LIN {X 54.744,Y 107.989,Z 76.139,A 180.000,B 0.000,C 180.000} C_DIS
LIN {X 54.880,Y 108.068,Z 76.134,A 180.000,B 0.000,C 180.000} C_DIS
LIN {X 55.020,Y 108.140,Z 76.129,A 180.000,B 0.000,C 180.000} C_DIS
LIN {X 55.161,Y 108.210,Z 76.124,A 180.000,B 0.000,C 180.000} C_DIS
LIN {X 55.302,Y 108.281,Z 76.120,A 180.000,B 0.000,C 180.000} C_DIS
LIN {X 55.444,Y 108.349,Z 76.115,A 180.000,B 0.000,C 180.000} C_DIS
LIN {X 55.590,Y 108.409,Z 76.111,A 180.000,B 0.000,C 180.000} C_DIS
LIN {X 55.736,Y 108.467,Z 76.106,A 180.000,B 0.000,C 180.000} C_DIS
LIN {X 55.883,Y 108.525,Z 76.102,A 180.000,B 0.000,C 180.000} C_DIS
LIN {X 56.030,Y 108.581,Z 76.097,A 180.000,B 0.000,C 180.000} C_DIS
LIN {X 56.180,Y 108.630,Z 76.093,A 180.000,B 0.000,C 180.000} C_DIS
LIN {X 56.331,Y 108.674,Z 76.089,A 180.000,B 0.000,C 180.000} C_DIS
LIN {X 56.482,Y 108.719,Z 76.085,A 180.000,B 0.000,C 180.000} C_DIS
LIN {X 56.633,Y 108.763,Z 76.081,A 180.000,B 0.000,C 180.000} C_DIS
LIN {X 56.786,Y 108.800,Z 76.077,A 180.000,B 0.000,C 180.000} C_DIS
LIN {X 56.940,Y 108.831,Z 76.073,A 180.000,B 0.000,C 180.000} C_DIS
LIN {X 57.095,Y 108.863,Z 76.070,A 180.000,B 0.000,C 180.000} C_DIS
LIN {X 57.249,Y 108.894,Z 76.066,A 180.000,B 0.000,C 180.000} C_DIS
LIN {X 57.405,Y 108.919,Z 76.062,A 180.000,B 0.000,C 180.000} C_DIS
LIN {X 57.561,Y 108.937,Z 76.059,A 180.000,B 0.000,C 180.000} C_DIS
LIN {X 57.718,Y 108.954,Z 76.056,A 180.000,B 0.000,C 180.000} C_DIS
LIN {X 57.874,Y 108.972,Z 76.052,A 180.000,B 0.000,C 180.000} C_DIS
LIN {X 58.031,Y 108.985,Z 76.049,A 180.000,B 0.000,C 180.000} C_DIS
LIN {X 58.188,Y 108.990,Z 76.046,A 180.000,B 0.000,C 180.000} C_DIS
LIN {X 58.346,Y 108.994,Z 76.043,A 180.000,B 0.000,C 180.000} C_DIS
LIN {X 58.503,Y 108.997,Z 76.040,A 180.000,B 0.000,C 180.000} C_DIS
LIN {X 58.661,Y 108.998,Z 76.037,A 180.000,B 0.000,C 180.000} C_DIS
LIN {X 58.818,Y 108.991,Z 76.034,A 180.000,B 0.000,C 180.000} C_DIS
LIN {X 58.975,Y 108.980,Z 76.032,A 180.000,B 0.000,C 180.000} C_DIS
LIN {X 59.132,Y 108.970,Z 76.029,A 180.000,B 0.000,C 180.000} C_DIS
LIN {X 59.290,Y 108.958,Z 76.027,A 180.000,B 0.000,C 180.000} C_DIS
LIN {X 59.601,Y 108.914,Z 76.022,A 180.000,B 0.000,C 180.000} C_DIS
LIN {X 59.913,Y 108.865,Z 76.018,A 180.000,B 0.000,C 180.000} C_DIS
LIN {X 60.220,Y 108.796,Z 76.014,A 180.000,B 0.000,C 180.000} C_DIS
LIN {X 60.526,Y 108.720,Z 76.011,A 180.000,B 0.000,C 180.000} C_DIS
LIN {X 60.826,Y 108.626,Z 76.008,A 180.000,B 0.000,C 180.000} C_DIS
LIN {X 61.124,Y 108.523,Z 76.005,A 180.000,B 0.000,C 180.000} C_DIS
LIN {X 61.272,Y 108.469,Z 76.004,A 180.000,B 0.000,C 180.000} C_DIS
LIN {X 61.416,Y 108.406,Z 76.003,A 180.000,B 0.000,C 180.000} C_DIS
LIN {X 61.704,Y 108.278,Z 76.002,A 180.000,B 0.000,C 180.000} C_DIS
LIN {X 61.847,Y 108.212,Z 76.001,A 180.000,B 0.000,C 180.000} C_DIS
LIN {X 61.986,Y 108.138,Z 76.001,A 180.000,B 0.000,C 180.000} C_DIS
LIN {X 62.261,Y 107.984,Z 76.000,A 180.000,B 0.000,C 180.000} C_DIS
LIN {X 62.461,Y 107.866,Z 76.000,A 180.000,B 0.000,C 180.000} C_DIS
; Cutting Move Starts
LIN {X 62.562,Y 107.802,Z 76.000,A 180.000,B 0.000,C 180.000} C_DIS
LIN {X 62.825,Y 107.623,Z 76.000,A 180.000,B 0.000,C 180.000} C_DIS
LIN {X 62.930,Y 107.551,Z 76.000,A 180.000,B 0.000,C 180.000} C_DIS
LIN {X 63.071,Y 107.444,Z 76.000,A 180.000,B 0.000,C 180.000} C_DIS
LIN {X 63.109,Y 107.413,Z 76.000,A 180.000,B 0.000,C 180.000} C_DIS
LIN {X 63.290,Y 107.265,Z 76.000,A 180.000,B 0.000,C 180.000} C_DIS
LIN {X 63.467,Y 107.120,Z 76.000,A 180.000,B 0.000,C 180.000} C_DIS
LIN {X 63.504,Y 107.086,Z 76.000,A 180.000,B 0.000,C 180.000} C_DIS
LIN {X 63.645,Y 106.952,Z 76.000,A 180.000,B 0.000,C 180.000} C_DIS
LIN {X 63.873,Y 106.729,Z 76.000,A 180.000,B 0.000,C 180.000} C_DIS
LIN {X 64.003,Y 106.596,Z 76.000,A 180.000,B 0.000,C 180.000} C_DIS
LIN {X 64.043,Y 106.550,Z 76.000,A 180.000,B 0.000,C 180.000} C_DIS
LIN {X 64.196,Y 106.371,Z 76.000,A 180.000,B 0.000,C 180.000} C_DIS
LIN {X 64.349,Y 106.193,Z 76.000,A 180.000,B 0.000,C 180.000} C_DIS
LIN {X 64.360,Y 106.179,Z 76.000,A 180.000,B 0.000,C 180.000} C_DIS
LIN {X 64.487,Y 106.014,Z 76.000,A 180.000,B 0.000,C 180.000} C_DIS
LIN {X 64.718,Y 105.690,Z 76.000,A 180.000,B 0.000,C 180.000} C_DIS
LIN {X 64.742,Y 105.656,Z 76.000,A 180.000,B 0.000,C 180.000} C_DIS
LIN {X 64.856,Y 105.477,Z 76.000,A 180.000,B 0.000,C 180.000} C_DIS
LIN {X 65.075,Y 105.104,Z 76.000,A 180.000,B 0.000,C 180.000} C_DIS
LIN {X 65.163,Y 104.941,Z 76.000,A 180.000,B 0.000,C 180.000} C_DIS
LIN {X 65.248,Y 104.762,Z 76.000,A 180.000,B 0.000,C 180.000} C_DIS
LIN {X 65.333,Y 104.584,Z 76.000,A 180.000,B 0.000,C 180.000} C_DIS
LIN {X 65.415,Y 104.405,Z 76.000,A 180.000,B 0.000,C 180.000} C_DIS
LIN {X 65.433,Y 104.360,Z 76.000,A 180.000,B 0.000,C 180.000} C_DIS
LIN {X 65.483,Y 104.226,Z 76.000,A 180.000,B 0.000,C 180.000} C_DIS
LIN {X 65.549,Y 104.047,Z 76.000,A 180.000,B 0.000,C 180.000} C_DIS
LIN {X 65.612,Y 103.878,Z 76.000,A 180.000,B 0.000,C 180.000} C_DIS
LIN {X 65.615,Y 103.869,Z 76.000,A 180.000,B 0.000,C 180.000} C_DIS
LIN {X 65.672,Y 103.690,Z 76.000,A 180.000,B 0.000,C 180.000} C_DIS
LIN {X 65.720,Y 103.511,Z 76.000,A 180.000,B 0.000,C 180.000} C_DIS
LIN {X 65.791,Y 103.253,Z 76.000,A 180.000,B 0.000,C 180.000} C_DIS
LIN {X 65.815,Y 103.153,Z 76.000,A 180.000,B 0.000,C 180.000} C_DIS
LIN {X 65.850,Y 102.975,Z 76.000,A 180.000,B 0.000,C 180.000} C_DIS
LIN {X 65.914,Y 102.617,Z 76.000,A 180.000,B 0.000,C 180.000} C_DIS
LIN {X 65.941,Y 102.438,Z 76.000,A 180.000,B 0.000,C 180.000} C_DIS
LIN {X 65.957,Y 102.260,Z 76.000,A 180.000,B 0.000,C 180.000} C_DIS
LIN {X 65.973,Y 102.081,Z 76.000,A 180.000,B 0.000,C 180.000} C_DIS
LIN {X 65.989,Y 101.902,Z 76.000,A 180.000,B 0.000,C 180.000} C_DIS
LIN {X 65.995,Y 101.723,Z 76.000,A 180.000,B 0.000,C 180.000} C_DIS
LIN {X 65.995,Y 101.366,Z 76.000,A 180.000,B 0.000,C 180.000} C_DIS
LIN {X 65.993,Y 101.187,Z 76.000,A 180.000,B 0.000,C 180.000} C_DIS
LIN {X 65.981,Y 101.008,Z 76.000,A 180.000,B 0.000,C 180.000} C_DIS
LIN {X 65.949,Y 100.651,Z 76.000,A 180.000,B 0.000,C 180.000} C_DIS
LIN {X 65.929,Y 100.472,Z 76.000,A 180.000,B 0.000,C 180.000} C_DIS
LIN {X 65.898,Y 100.293,Z 76.000,A 180.000,B 0.000,C 180.000} C_DIS
LIN {X 65.866,Y 100.114,Z 76.000,A 180.000,B 0.000,C 180.000} C_DIS
LIN {X 65.834,Y 99.936,Z 76.000,A 180.000,B 0.000,C 180.000} C_DIS
LIN {X 65.793,Y 99.757,Z 76.000,A 180.000,B 0.000,C 180.000} C_DIS
LIN {X 65.791,Y 99.747,Z 76.000,A 180.000,B 0.000,C 180.000} C_DIS
LIN {X 65.696,Y 99.399,Z 76.000,A 180.000,B 0.000,C 180.000} C_DIS
LIN {X 65.645,Y 99.221,Z 76.000,A 180.000,B 0.000,C 180.000} C_DIS
LIN {X 65.612,Y 99.122,Z 76.000,A 180.000,B 0.000,C 180.000} C_DIS
LIN {X 65.582,Y 99.042,Z 76.000,A 180.000,B 0.000,C 180.000} C_DIS
LIN {X 65.516,Y 98.863,Z 76.000,A 180.000,B 0.000,C 180.000} C_DIS
LIN {X 65.450,Y 98.684,Z 76.000,A 180.000,B 0.000,C 180.000} C_DIS
LIN {X 65.433,Y 98.640,Z 76.000,A 180.000,B 0.000,C 180.000} C_DIS
LIN {X 65.375,Y 98.505,Z 76.000,A 180.000,B 0.000,C 180.000} C_DIS
LIN {X 65.290,Y 98.327,Z 76.000,A 180.000,B 0.000,C 180.000} C_DIS
LIN {X 65.206,Y 98.148,Z 76.000,A 180.000,B 0.000,C 180.000} C_DIS
LIN {X 65.117,Y 97.969,Z 76.000,A 180.000,B 0.000,C 180.000} C_DIS
LIN {X 65.075,Y 97.896,Z 76.000,A 180.000,B 0.000,C 180.000} C_DIS
LIN {X 64.897,Y 97.592,Z 76.000,A 180.000,B 0.000,C 180.000} C_DIS
LIN {X 64.801,Y 97.433,Z 76.000,A 180.000,B 0.000,C 180.000} C_DIS
LIN {X 64.718,Y 97.310,Z 76.000,A 180.000,B 0.000,C 180.000} C_DIS
LIN {X 64.539,Y 97.060,Z 76.000,A 180.000,B 0.000,C 180.000} C_DIS
LIN {X 64.421,Y 96.897,Z 76.000,A 180.000,B 0.000,C 180.000} C_DIS
LIN {X 64.360,Y 96.821,Z 76.000,A 180.000,B 0.000,C 180.000} C_DIS
LIN {X 64.272,Y 96.718,Z 76.000,A 180.000,B 0.000,C 180.000} C_DIS
LIN {X 64.119,Y 96.539,Z 76.000,A 180.000,B 0.000,C 180.000} C_DIS
LIN {X 64.003,Y 96.404,Z 76.000,A 180.000,B 0.000,C 180.000} C_DIS
LIN {X 63.962,Y 96.360,Z 76.000,A 180.000,B 0.000,C 180.000} C_DIS
LIN {X 63.824,Y 96.223,Z 76.000,A 180.000,B 0.000,C 180.000} C_DIS
LIN {X 63.599,Y 96.003,Z 76.000,A 180.000,B 0.000,C 180.000} C_DIS
LIN {X 63.467,Y 95.880,Z 76.000,A 180.000,B 0.000,C 180.000} C_DIS
LIN {X 63.399,Y 95.824,Z 76.000,A 180.000,B 0.000,C 180.000} C_DIS
LIN {X 63.109,Y 95.587,Z 76.000,A 180.000,B 0.000,C 180.000} C_DIS
LIN {X 62.954,Y 95.466,Z 76.000,A 180.000,B 0.000,C 180.000} C_DIS
LIN {X 62.930,Y 95.449,Z 76.000,A 180.000,B 0.000,C 180.000} C_DIS
LIN {X 62.751,Y 95.327,Z 76.000,A 180.000,B 0.000,C 180.000} C_DIS
LIN {X 62.573,Y 95.206,Z 76.000,A 180.000,B 0.000,C 180.000} C_DIS
LIN {X 62.425,Y 95.109,Z 76.000,A 180.000,B 0.000,C 180.000} C_DIS
LIN {X 62.394,Y 95.091,Z 76.000,A 180.000,B 0.000,C 180.000} C_DIS
LIN {X 62.215,Y 94.990,Z 76.000,A 180.000,B 0.000,C 180.000} C_DIS
LIN {X 62.036,Y 94.890,Z 76.000,A 180.000,B 0.000,C 180.000} C_DIS
LIN {X 61.858,Y 94.794,Z 76.000,A 180.000,B 0.000,C 180.000} C_DIS
LIN {X 61.769,Y 94.751,Z 76.000,A 180.000,B 0.000,C 180.000} C_DIS
LIN {X 61.679,Y 94.711,Z 76.000,A 180.000,B 0.000,C 180.000} C_DIS
LIN {X 61.369,Y 94.573,Z 76.000,A 180.000,B 0.000,C 180.000} C_DIS
LIN {X 61.321,Y 94.552,Z 76.000,A 180.000,B 0.000,C 180.000} C_DIS
LIN {X 61.143,Y 94.483,Z 76.000,A 180.000,B 0.000,C 180.000} C_DIS
LIN {X 60.785,Y 94.360,Z 76.000,A 180.000,B 0.000,C 180.000} C_DIS
LIN {X 60.606,Y 94.302,Z 76.000,A 180.000,B 0.000,C 180.000} C_DIS
LIN {X 60.427,Y 94.256,Z 76.000,A 180.000,B 0.000,C 180.000} C_DIS
LIN {X 60.249,Y 94.212,Z 76.000,A 180.000,B 0.000,C 180.000} C_DIS
LIN {X 60.070,Y 94.167,Z 76.000,A 180.000,B 0.000,C 180.000} C_DIS
LIN {X 59.891,Y 94.131,Z 76.000,A 180.000,B 0.000,C 180.000} C_DIS
LIN {X 59.712,Y 94.103,Z 76.000,A 180.000,B 0.000,C 180.000} C_DIS
LIN {X 59.534,Y 94.075,Z 76.000,A 180.000,B 0.000,C 180.000} C_DIS
LIN {X 59.355,Y 94.049,Z 76.000,A 180.000,B 0.000,C 180.000} C_DIS
LIN {X 59.220,Y 94.036,Z 76.000,A 180.000,B 0.000,C 180.000} C_DIS
LIN {X 58.819,Y 94.010,Z 76.000,A 180.000,B 0.000,C 180.000} C_DIS
LIN {X 58.640,Y 94.001,Z 76.000,A 180.000,B 0.000,C 180.000} C_DIS
LIN {X 58.461,Y 94.004,Z 76.000,A 180.000,B 0.000,C 180.000} C_DIS
LIN {X 58.282,Y 94.008,Z 76.000,A 180.000,B 0.000,C 180.000} C_DIS
LIN {X 58.103,Y 94.012,Z 76.000,A 180.000,B 0.000,C 180.000} C_DIS
LIN {X 57.925,Y 94.023,Z 76.000,A 180.000,B 0.000,C 180.000} C_DIS
LIN {X 57.803,Y 94.036,Z 76.000,A 180.000,B 0.000,C 180.000} C_DIS
LIN {X 57.567,Y 94.062,Z 76.000,A 180.000,B 0.000,C 180.000} C_DIS
LIN {X 57.388,Y 94.083,Z 76.000,A 180.000,B 0.000,C 180.000} C_DIS
LIN {X 57.210,Y 94.114,Z 76.000,A 180.000,B 0.000,C 180.000} C_DIS
LIN {X 56.852,Y 94.186,Z 76.000,A 180.000,B 0.000,C 180.000} C_DIS
LIN {X 56.717,Y 94.215,Z 76.000,A 180.000,B 0.000,C 180.000} C_DIS
LIN {X 56.673,Y 94.226,Z 76.000,A 180.000,B 0.000,C 180.000} C_DIS
LIN {X 56.495,Y 94.277,Z 76.000,A 180.000,B 0.000,C 180.000} C_DIS
LIN {X 56.316,Y 94.330,Z 76.000,A 180.000,B 0.000,C 180.000} C_DIS
LIN {X 56.137,Y 94.383,Z 76.000,A 180.000,B 0.000,C 180.000} C_DIS
LIN {X 56.103,Y 94.394,Z 76.000,A 180.000,B 0.000,C 180.000} C_DIS
LIN {X 55.958,Y 94.445,Z 76.000,A 180.000,B 0.000,C 180.000} C_DIS
LIN {X 55.601,Y 94.587,Z 76.000,A 180.000,B 0.000,C 180.000} C_DIS
LIN {X 55.422,Y 94.661,Z 76.000,A 180.000,B 0.000,C 180.000} C_DIS
LIN {X 55.243,Y 94.749,Z 76.000,A 180.000,B 0.000,C 180.000} C_DIS
LIN {X 55.064,Y 94.838,Z 76.000,A 180.000,B 0.000,C 180.000} C_DIS
LIN {X 54.886,Y 94.929,Z 76.000,A 180.000,B 0.000,C 180.000} C_DIS
LIN {X 54.883,Y 94.930,Z 76.000,A 180.000,B 0.000,C 180.000} C_DIS
LIN {X 54.707,Y 95.033,Z 76.000,A 180.000,B 0.000,C 180.000} C_DIS
LIN {X 54.528,Y 95.144,Z 76.000,A 180.000,B 0.000,C 180.000} C_DIS
LIN {X 54.349,Y 95.254,Z 76.000,A 180.000,B 0.000,C 180.000} C_DIS
LIN {X 54.298,Y 95.288,Z 76.000,A 180.000,B 0.000,C 180.000} C_DIS
LIN {X 54.171,Y 95.379,Z 76.000,A 180.000,B 0.000,C 180.000} C_DIS
LIN {X 53.992,Y 95.512,Z 76.000,A 180.000,B 0.000,C 180.000} C_DIS
LIN {X 53.814,Y 95.645,Z 76.000,A 180.000,B 0.000,C 180.000} C_DIS
LIN {X 53.813,Y 95.646,Z 76.000,A 180.000,B 0.000,C 180.000} C_DIS
LIN {X 53.634,Y 95.796,Z 76.000,A 180.000,B 0.000,C 180.000} C_DIS
LIN {X 53.404,Y 96.003,Z 76.000,A 180.000,B 0.000,C 180.000} C_DIS
LIN {X 53.277,Y 96.118,Z 76.000,A 180.000,B 0.000,C 180.000} C_DIS
LIN {X 53.213,Y 96.181,Z 76.000,A 180.000,B 0.000,C 180.000} C_DIS
LIN {X 53.098,Y 96.303,Z 76.000,A 180.000,B 0.000,C 180.000} C_DIS
LIN {X 52.877,Y 96.539,Z 76.000,A 180.000,B 0.000,C 180.000} C_DIS
LIN {X 52.740,Y 96.698,Z 76.000,A 180.000,B 0.000,C 180.000} C_DIS
LIN {X 52.725,Y 96.718,Z 76.000,A 180.000,B 0.000,C 180.000} C_DIS
LIN {X 52.562,Y 96.927,Z 76.000,A 180.000,B 0.000,C 180.000} C_DIS
LIN {X 52.446,Y 97.075,Z 76.000,A 180.000,B 0.000,C 180.000} C_DIS
LIN {X 52.383,Y 97.161,Z 76.000,A 180.000,B 0.000,C 180.000} C_DIS
LIN {X 52.320,Y 97.254,Z 76.000,A 180.000,B 0.000,C 180.000} C_DIS
LIN {X 52.088,Y 97.612,Z 76.000,A 180.000,B 0.000,C 180.000} C_DIS
LIN {X 52.025,Y 97.715,Z 76.000,A 180.000,B 0.000,C 180.000} C_DIS
LIN {X 51.983,Y 97.790,Z 76.000,A 180.000,B 0.000,C 180.000} C_DIS
LIN {X 51.889,Y 97.969,Z 76.000,A 180.000,B 0.000,C 180.000} C_DIS
LIN {X 51.794,Y 98.148,Z 76.000,A 180.000,B 0.000,C 180.000} C_DIS
LIN {X 51.705,Y 98.327,Z 76.000,A 180.000,B 0.000,C 180.000} C_DIS
LIN {X 51.668,Y 98.412,Z 76.000,A 180.000,B 0.000,C 180.000} C_DIS
LIN {X 51.553,Y 98.684,Z 76.000,A 180.000,B 0.000,C 180.000} C_DIS
LIN {X 51.489,Y 98.838,Z 76.000,A 180.000,B 0.000,C 180.000} C_DIS
LIN {X 51.479,Y 98.863,Z 76.000,A 180.000,B 0.000,C 180.000} C_DIS
LIN {X 51.417,Y 99.042,Z 76.000,A 180.000,B 0.000,C 180.000} C_DIS
LIN {X 51.303,Y 99.399,Z 76.000,A 180.000,B 0.000,C 180.000} C_DIS
LIN {X 51.251,Y 99.578,Z 76.000,A 180.000,B 0.000,C 180.000} C_DIS
LIN {X 51.210,Y 99.757,Z 76.000,A 180.000,B 0.000,C 180.000} C_DIS
LIN {X 51.170,Y 99.936,Z 76.000,A 180.000,B 0.000,C 180.000} C_DIS
LIN {X 51.131,Y 100.106,Z 76.000,A 180.000,B 0.000,C 180.000} C_DIS
LIN {X 51.130,Y 100.114,Z 76.000,A 180.000,B 0.000,C 180.000} C_DIS
LIN {X 51.100,Y 100.293,Z 76.000,A 180.000,B 0.000,C 180.000} C_DIS
LIN {X 51.052,Y 100.651,Z 76.000,A 180.000,B 0.000,C 180.000} C_DIS
LIN {X 51.030,Y 100.829,Z 76.000,A 180.000,B 0.000,C 180.000} C_DIS
LIN {X 51.019,Y 101.008,Z 76.000,A 180.000,B 0.000,C 180.000} C_DIS
LIN {X 51.003,Y 101.366,Z 76.000,A 180.000,B 0.000,C 180.000} C_DIS
LIN {X 51.000,Y 101.545,Z 76.000,A 180.000,B 0.000,C 180.000} C_DIS
LIN {X 51.007,Y 101.723,Z 76.000,A 180.000,B 0.000,C 180.000} C_DIS
LIN {X 51.015,Y 101.902,Z 76.000,A 180.000,B 0.000,C 180.000} C_DIS
LIN {X 51.023,Y 102.081,Z 76.000,A 180.000,B 0.000,C 180.000} C_DIS
LIN {X 51.040,Y 102.260,Z 76.000,A 180.000,B 0.000,C 180.000} C_DIS
LIN {X 51.064,Y 102.438,Z 76.000,A 180.000,B 0.000,C 180.000} C_DIS
LIN {X 51.088,Y 102.617,Z 76.000,A 180.000,B 0.000,C 180.000} C_DIS
LIN {X 51.113,Y 102.796,Z 76.000,A 180.000,B 0.000,C 180.000} C_DIS
LIN {X 51.131,Y 102.894,Z 76.000,A 180.000,B 0.000,C 180.000} C_DIS
LIN {X 51.149,Y 102.975,Z 76.000,A 180.000,B 0.000,C 180.000} C_DIS
LIN {X 51.230,Y 103.332,Z 76.000,A 180.000,B 0.000,C 180.000} C_DIS
LIN {X 51.275,Y 103.511,Z 76.000,A 180.000,B 0.000,C 180.000} C_DIS
LIN {X 51.310,Y 103.624,Z 76.000,A 180.000,B 0.000,C 180.000} C_DIS
LIN {X 51.388,Y 103.869,Z 76.000,A 180.000,B 0.000,C 180.000} C_DIS
LIN {X 51.446,Y 104.047,Z 76.000,A 180.000,B 0.000,C 180.000} C_DIS
LIN {X 51.489,Y 104.162,Z 76.000,A 180.000,B 0.000,C 180.000} C_DIS
LIN {X 51.515,Y 104.226,Z 76.000,A 180.000,B 0.000,C 180.000} C_DIS
LIN {X 51.668,Y 104.588,Z 76.000,A 180.000,B 0.000,C 180.000} C_DIS
LIN {X 51.747,Y 104.762,Z 76.000,A 180.000,B 0.000,C 180.000} C_DIS
LIN {X 51.841,Y 104.941,Z 76.000,A 180.000,B 0.000,C 180.000} C_DIS
LIN {X 51.936,Y 105.120,Z 76.000,A 180.000,B 0.000,C 180.000} C_DIS
LIN {X 52.025,Y 105.285,Z 76.000,A 180.000,B 0.000,C 180.000} C_DIS
LIN {X 52.033,Y 105.299,Z 76.000,A 180.000,B 0.000,C 180.000} C_DIS
LIN {X 52.146,Y 105.477,Z 76.000,A 180.000,B 0.000,C 180.000} C_DIS
LIN {X 52.262,Y 105.656,Z 76.000,A 180.000,B 0.000,C 180.000} C_DIS
LIN {X 52.380,Y 105.835,Z 76.000,A 180.000,B 0.000,C 180.000} C_DIS
LIN {X 52.383,Y 105.839,Z 76.000,A 180.000,B 0.000,C 180.000} C_DIS
LIN {X 52.515,Y 106.014,Z 76.000,A 180.000,B 0.000,C 180.000} C_DIS
LIN {X 52.655,Y 106.193,Z 76.000,A 180.000,B 0.000,C 180.000} C_DIS
LIN {X 52.740,Y 106.302,Z 76.000,A 180.000,B 0.000,C 180.000} C_DIS
LIN {X 52.797,Y 106.371,Z 76.000,A 180.000,B 0.000,C 180.000} C_DIS
LIN {X 52.919,Y 106.506,Z 76.000,A 180.000,B 0.000,C 180.000} C_DIS
LIN {X 53.128,Y 106.729,Z 76.000,A 180.000,B 0.000,C 180.000} C_DIS
LIN {X 53.277,Y 106.882,Z 76.000,A 180.000,B 0.000,C 180.000} C_DIS
LIN {X 53.304,Y 106.908,Z 76.000,A 180.000,B 0.000,C 180.000} C_DIS
LIN {X 53.455,Y 107.044,Z 76.000,A 180.000,B 0.000,C 180.000} C_DIS
LIN {X 53.634,Y 107.204,Z 76.000,A 180.000,B 0.000,C 180.000} C_DIS
LIN {X 53.704,Y 107.265,Z 76.000,A 180.000,B 0.000,C 180.000} C_DIS
LIN {X 53.813,Y 107.354,Z 76.000,A 180.000,B 0.000,C 180.000} C_DIS
LIN {X 53.933,Y 107.444,Z 76.000,A 180.000,B 0.000,C 180.000} C_DIS
LIN {X 54.172,Y 107.623,Z 76.000,A 180.000,B 0.000,C 180.000} C_DIS
LIN {X 54.349,Y 107.746,Z 76.000,A 180.000,B 0.000,C 180.000} C_DIS
LIN {X 54.439,Y 107.802,Z 76.000,A 180.000,B 0.000,C 180.000} C_DIS
LIN {X 54.729,Y 107.980,Z 76.000,A 180.000,B 0.000,C 180.000} C_DIS
LIN {X 54.886,Y 108.071,Z 76.000,A 180.000,B 0.000,C 180.000} C_DIS
LIN {X 55.059,Y 108.159,Z 76.000,A 180.000,B 0.000,C 180.000} C_DIS
LIN {X 55.243,Y 108.251,Z 76.000,A 180.000,B 0.000,C 180.000} C_DIS
LIN {X 55.419,Y 108.338,Z 76.000,A 180.000,B 0.000,C 180.000} C_DIS
LIN {X 55.422,Y 108.339,Z 76.000,A 180.000,B 0.000,C 180.000} C_DIS
LIN {X 55.601,Y 108.413,Z 76.000,A 180.000,B 0.000,C 180.000} C_DIS
LIN {X 55.862,Y 108.517,Z 76.000,A 180.000,B 0.000,C 180.000} C_DIS
LIN {X 55.958,Y 108.555,Z 76.000,A 180.000,B 0.000,C 180.000} C_DIS
LIN {X 56.137,Y 108.617,Z 76.000,A 180.000,B 0.000,C 180.000} C_DIS
LIN {X 56.316,Y 108.670,Z 76.000,A 180.000,B 0.000,C 180.000} C_DIS
LIN {X 56.495,Y 108.723,Z 76.000,A 180.000,B 0.000,C 180.000} C_DIS
LIN {X 56.673,Y 108.774,Z 76.000,A 180.000,B 0.000,C 180.000} C_DIS
LIN {X 56.852,Y 108.814,Z 76.000,A 180.000,B 0.000,C 180.000} C_DIS
LIN {X 57.210,Y 108.886,Z 76.000,A 180.000,B 0.000,C 180.000} C_DIS
LIN {X 57.388,Y 108.917,Z 76.000,A 180.000,B 0.000,C 180.000} C_DIS
LIN {X 57.567,Y 108.938,Z 76.000,A 180.000,B 0.000,C 180.000} C_DIS
LIN {X 57.746,Y 108.957,Z 76.000,A 180.000,B 0.000,C 180.000} C_DIS
LIN {X 57.925,Y 108.977,Z 76.000,A 180.000,B 0.000,C 180.000} C_DIS
LIN {X 58.103,Y 108.988,Z 76.000,A 180.000,B 0.000,C 180.000} C_DIS
LIN {X 58.282,Y 108.992,Z 76.000,A 180.000,B 0.000,C 180.000} C_DIS
LIN {X 58.461,Y 108.996,Z 76.000,A 180.000,B 0.000,C 180.000} C_DIS
LIN {X 58.640,Y 108.999,Z 76.000,A 180.000,B 0.000,C 180.000} C_DIS
LIN {X 58.819,Y 108.990,Z 76.000,A 180.000,B 0.000,C 180.000} C_DIS
LIN {X 59.176,Y 108.967,Z 76.000,A 180.000,B 0.000,C 180.000} C_DIS
LIN {X 59.355,Y 108.951,Z 76.000,A 180.000,B 0.000,C 180.000} C_DIS
LIN {X 59.534,Y 108.925,Z 76.000,A 180.000,B 0.000,C 180.000} C_DIS
LIN {X 59.856,Y 108.874,Z 76.000,A 180.000,B 0.000,C 180.000} C_DIS
LIN {X 59.891,Y 108.869,Z 76.000,A 180.000,B 0.000,C 180.000} C_DIS
LIN {X 60.070,Y 108.833,Z 76.000,A 180.000,B 0.000,C 180.000} C_DIS
LIN {X 60.249,Y 108.788,Z 76.000,A 180.000,B 0.000,C 180.000} C_DIS
LIN {X 60.427,Y 108.744,Z 76.000,A 180.000,B 0.000,C 180.000} C_DIS
LIN {X 60.606,Y 108.698,Z 76.000,A 180.000,B 0.000,C 180.000} C_DIS
LIN {X 60.616,Y 108.695,Z 76.000,A 180.000,B 0.000,C 180.000} C_DIS
LIN {X 60.785,Y 108.640,Z 76.000,A 180.000,B 0.000,C 180.000} C_DIS
LIN {X 61.144,Y 108.517,Z 76.000,A 180.000,B 0.000,C 180.000} C_DIS
LIN {X 61.321,Y 108.448,Z 76.000,A 180.000,B 0.000,C 180.000} C_DIS
LIN {X 61.500,Y 108.369,Z 76.000,A 180.000,B 0.000,C 180.000} C_DIS
LIN {X 61.679,Y 108.289,Z 76.000,A 180.000,B 0.000,C 180.000} C_DIS
LIN {X 61.858,Y 108.206,Z 76.000,A 180.000,B 0.000,C 180.000} C_DIS
LIN {X 61.948,Y 108.159,Z 76.000,A 180.000,B 0.000,C 180.000} C_DIS
LIN {X 62.036,Y 108.110,Z 76.000,A 180.000,B 0.000,C 180.000} C_DIS
LIN {X 62.268,Y 107.980,Z 76.000,A 180.000,B 0.000,C 180.000} C_DIS
LIN {X 62.394,Y 107.909,Z 76.000,A 180.000,B 0.000,C 180.000} C_DIS
LIN {X 62.461,Y 107.866,Z 76.000,A 180.000,B 0.000,C 180.000} C_DIS
; Link Move Starts
LIN {X 62.724,Y 107.692,Z 76.000,A 180.000,B 0.000,C 180.000} C_DIS
LIN {X 62.983,Y 107.513,Z 75.999,A 180.000,B 0.000,C 180.000} C_DIS
LIN {X 63.228,Y 107.315,Z 75.998,A 180.000,B 0.000,C 180.000} C_DIS
LIN {X 63.472,Y 107.115,Z 75.996,A 180.000,B 0.000,C 180.000} C_DIS
LIN {X 63.700,Y 106.898,Z 75.994,A 180.000,B 0.000,C 180.000} C_DIS
LIN {X 63.925,Y 106.678,Z 75.991,A 180.000,B 0.000,C 180.000} C_DIS
LIN {X 64.135,Y 106.443,Z 75.988,A 180.000,B 0.000,C 180.000} C_DIS
LIN {X 64.340,Y 106.204,Z 75.985,A 180.000,B 0.000,C 180.000} C_DIS
LIN {X 64.438,Y 106.081,Z 75.983,A 180.000,B 0.000,C 180.000} C_DIS
LIN {X 64.530,Y 105.953,Z 75.981,A 180.000,B 0.000,C 180.000} C_DIS
LIN {X 64.713,Y 105.697,Z 75.977,A 180.000,B 0.000,C 180.000} C_DIS
LIN {X 64.802,Y 105.566,Z 75.974,A 180.000,B 0.000,C 180.000} C_DIS
LIN {X 64.883,Y 105.431,Z 75.972,A 180.000,B 0.000,C 180.000} C_DIS
LIN {X 64.963,Y 105.296,Z 75.969,A 180.000,B 0.000,C 180.000} C_DIS
LIN {X 65.043,Y 105.160,Z 75.967,A 180.000,B 0.000,C 180.000} C_DIS
LIN {X 65.121,Y 105.023,Z 75.964,A 180.000,B 0.000,C 180.000} C_DIS
LIN {X 65.191,Y 104.882,Z 75.961,A 180.000,B 0.000,C 180.000} C_DIS
LIN {X 65.259,Y 104.740,Z 75.959,A 180.000,B 0.000,C 180.000} C_DIS
LIN {X 65.326,Y 104.598,Z 75.956,A 180.000,B 0.000,C 180.000} C_DIS
LIN {X 65.393,Y 104.455,Z 75.952,A 180.000,B 0.000,C 180.000} C_DIS
LIN {X 65.452,Y 104.309,Z 75.949,A 180.000,B 0.000,C 180.000} C_DIS
LIN {X 65.507,Y 104.161,Z 75.946,A 180.000,B 0.000,C 180.000} C_DIS
LIN {X 65.562,Y 104.014,Z 75.943,A 180.000,B 0.000,C 180.000} C_DIS
LIN {X 65.616,Y 103.866,Z 75.939,A 180.000,B 0.000,C 180.000} C_DIS
LIN {X 65.664,Y 103.716,Z 75.936,A 180.000,B 0.000,C 180.000} C_DIS
LIN {X 65.706,Y 103.564,Z 75.932,A 180.000,B 0.000,C 180.000} C_DIS
LIN {X 65.747,Y 103.412,Z 75.928,A 180.000,B 0.000,C 180.000} C_DIS
LIN {X 65.789,Y 103.260,Z 75.925,A 180.000,B 0.000,C 180.000} C_DIS
LIN {X 65.826,Y 103.107,Z 75.921,A 180.000,B 0.000,C 180.000} C_DIS
LIN {X 65.854,Y 102.952,Z 75.917,A 180.000,B 0.000,C 180.000} C_DIS
LIN {X 65.882,Y 102.797,Z 75.913,A 180.000,B 0.000,C 180.000} C_DIS
LIN {X 65.910,Y 102.642,Z 75.909,A 180.000,B 0.000,C 180.000} C_DIS
LIN {X 65.935,Y 102.487,Z 75.905,A 180.000,B 0.000,C 180.000} C_DIS
LIN {X 65.951,Y 102.330,Z 75.900,A 180.000,B 0.000,C 180.000} C_DIS
LIN {X 65.965,Y 102.173,Z 75.896,A 180.000,B 0.000,C 180.000} C_DIS
LIN {X 65.979,Y 102.016,Z 75.892,A 180.000,B 0.000,C 180.000} C_DIS
LIN {X 65.991,Y 101.859,Z 75.887,A 180.000,B 0.000,C 180.000} C_DIS
LIN {X 65.995,Y 101.702,Z 75.883,A 180.000,B 0.000,C 180.000} C_DIS
LIN {X 65.995,Y 101.544,Z 75.878,A 180.000,B 0.000,C 180.000} C_DIS
LIN {X 65.995,Y 101.387,Z 75.873,A 180.000,B 0.000,C 180.000} C_DIS
LIN {X 65.995,Y 101.229,Z 75.869,A 180.000,B 0.000,C 180.000} C_DIS
LIN {X 65.987,Y 101.072,Z 75.864,A 180.000,B 0.000,C 180.000} C_DIS
LIN {X 65.973,Y 100.915,Z 75.859,A 180.000,B 0.000,C 180.000} C_DIS
LIN {X 65.959,Y 100.758,Z 75.854,A 180.000,B 0.000,C 180.000} C_DIS
LIN {X 65.952,Y 100.680,Z 75.851,A 180.000,B 0.000,C 180.000} C_DIS
LIN {X 65.945,Y 100.601,Z 75.849,A 180.000,B 0.000,C 180.000} C_DIS
LIN {X 65.936,Y 100.523,Z 75.846,A 180.000,B 0.000,C 180.000} C_DIS
LIN {X 65.925,Y 100.445,Z 75.844,A 180.000,B 0.000,C 180.000} C_DIS
LIN {X 65.911,Y 100.367,Z 75.841,A 180.000,B 0.000,C 180.000} C_DIS
LIN {X 65.898,Y 100.290,Z 75.839,A 180.000,B 0.000,C 180.000} C_DIS
LIN {X 65.884,Y 100.212,Z 75.836,A 180.000,B 0.000,C 180.000} C_DIS
LIN {X 65.856,Y 100.057,Z 75.831,A 180.000,B 0.000,C 180.000} C_DIS
LIN {X 65.842,Y 99.980,Z 75.828,A 180.000,B 0.000,C 180.000} C_DIS
LIN {X 65.828,Y 99.902,Z 75.825,A 180.000,B 0.000,C 180.000} C_DIS
LIN {X 65.811,Y 99.825,Z 75.823,A 180.000,B 0.000,C 180.000} C_DIS
LIN {X 65.791,Y 99.749,Z 75.820,A 180.000,B 0.000,C 180.000} C_DIS
LIN {X 65.750,Y 99.597,Z 75.815,A 180.000,B 0.000,C 180.000} C_DIS
LIN {X 65.709,Y 99.445,Z 75.809,A 180.000,B 0.000,C 180.000} C_DIS
LIN {X 65.688,Y 99.369,Z 75.807,A 180.000,B 0.000,C 180.000} C_DIS
LIN {X 65.667,Y 99.293,Z 75.804,A 180.000,B 0.000,C 180.000} C_DIS
LIN {X 65.644,Y 99.218,Z 75.801,A 180.000,B 0.000,C 180.000} C_DIS
LIN {X 65.619,Y 99.143,Z 75.798,A 180.000,B 0.000,C 180.000} C_DIS
LIN {X 65.592,Y 99.069,Z 75.796,A 180.000,B 0.000,C 180.000} C_DIS
LIN {X 65.538,Y 98.921,Z 75.790,A 180.000,B 0.000,C 180.000} C_DIS
LIN {X 65.456,Y 98.700,Z 75.782,A 180.000,B 0.000,C 180.000} C_DIS
LIN {X 65.427,Y 98.626,Z 75.779,A 180.000,B 0.000,C 180.000} C_DIS
LIN {X 65.397,Y 98.554,Z 75.776,A 180.000,B 0.000,C 180.000} C_DIS
LIN {X 65.364,Y 98.482,Z 75.774,A 180.000,B 0.000,C 180.000} C_DIS
LIN {X 65.297,Y 98.340,Z 75.768,A 180.000,B 0.000,C 180.000} C_DIS
LIN {X 65.195,Y 98.126,Z 75.760,A 180.000,B 0.000,C 180.000} C_DIS
LIN {X 65.161,Y 98.055,Z 75.757,A 180.000,B 0.000,C 180.000} C_DIS
LIN {X 65.125,Y 97.985,Z 75.754,A 180.000,B 0.000,C 180.000} C_DIS
LIN {X 65.087,Y 97.916,Z 75.752,A 180.000,B 0.000,C 180.000} C_DIS
LIN {X 65.048,Y 97.848,Z 75.749,A 180.000,B 0.000,C 180.000} C_DIS
LIN {X 64.968,Y 97.713,Z 75.743,A 180.000,B 0.000,C 180.000} C_DIS
LIN {X 64.928,Y 97.645,Z 75.741,A 180.000,B 0.000,C 180.000} C_DIS
LIN {X 64.848,Y 97.509,Z 75.735,A 180.000,B 0.000,C 180.000} C_DIS
LIN {X 64.807,Y 97.442,Z 75.732,A 180.000,B 0.000,C 180.000} C_DIS
LIN {X 64.764,Y 97.376,Z 75.730,A 180.000,B 0.000,C 180.000} C_DIS
LIN {X 64.719,Y 97.311,Z 75.727,A 180.000,B 0.000,C 180.000} C_DIS
LIN {X 64.627,Y 97.183,Z 75.721,A 180.000,B 0.000,C 180.000} C_DIS
LIN {X 64.581,Y 97.119,Z 75.719,A 180.000,B 0.000,C 180.000} C_DIS
LIN {X 64.490,Y 96.991,Z 75.713,A 180.000,B 0.000,C 180.000} C_DIS
LIN {X 64.444,Y 96.927,Z 75.710,A 180.000,B 0.000,C 180.000} C_DIS
LIN {X 64.396,Y 96.864,Z 75.708,A 180.000,B 0.000,C 180.000} C_DIS
LIN {X 64.346,Y 96.804,Z 75.705,A 180.000,B 0.000,C 180.000} C_DIS
LIN {X 64.295,Y 96.744,Z 75.702,A 180.000,B 0.000,C 180.000} C_DIS
LIN {X 64.090,Y 96.504,Z 75.691,A 180.000,B 0.000,C 180.000} C_DIS
LIN {X 64.039,Y 96.445,Z 75.688,A 180.000,B 0.000,C 180.000} C_DIS
LIN {X 63.986,Y 96.386,Z 75.686,A 180.000,B 0.000,C 180.000} C_DIS
LIN {X 63.932,Y 96.329,Z 75.683,A 180.000,B 0.000,C 180.000} C_DIS
LIN {X 63.876,Y 96.274,Z 75.680,A 180.000,B 0.000,C 180.000} C_DIS
LIN {X 63.594,Y 95.998,Z 75.666,A 180.000,B 0.000,C 180.000} C_DIS
LIN {X 63.537,Y 95.944,Z 75.664,A 180.000,B 0.000,C 180.000} C_DIS
LIN {X 63.479,Y 95.891,Z 75.661,A 180.000,B 0.000,C 180.000} C_DIS
LIN {X 63.419,Y 95.840,Z 75.658,A 180.000,B 0.000,C 180.000} C_DIS
LIN {X 63.114,Y 95.591,Z 75.644,A 180.000,B 0.000,C 180.000} C_DIS
LIN {X 63.053,Y 95.541,Z 75.642,A 180.000,B 0.000,C 180.000} C_DIS
LIN {X 62.991,Y 95.493,Z 75.639,A 180.000,B 0.000,C 180.000} C_DIS
LIN {X 62.927,Y 95.447,Z 75.636,A 180.000,B 0.000,C 180.000} C_DIS
LIN {X 62.862,Y 95.402,Z 75.633,A 180.000,B 0.000,C 180.000} C_DIS
LIN {X 62.732,Y 95.314,Z 75.628,A 180.000,B 0.000,C 180.000} C_DIS
LIN {X 62.536,Y 95.181,Z 75.620,A 180.000,B 0.000,C 180.000} C_DIS
LIN {X 62.471,Y 95.137,Z 75.617,A 180.000,B 0.000,C 180.000} C_DIS
LIN {X 62.403,Y 95.096,Z 75.614,A 180.000,B 0.000,C 180.000} C_DIS
LIN {X 62.335,Y 95.057,Z 75.611,A 180.000,B 0.000,C 180.000} C_DIS
LIN {X 62.129,Y 94.942,Z 75.603,A 180.000,B 0.000,C 180.000} C_DIS
LIN {X 61.991,Y 94.865,Z 75.598,A 180.000,B 0.000,C 180.000} C_DIS
LIN {X 61.922,Y 94.827,Z 75.595,A 180.000,B 0.000,C 180.000} C_DIS
LIN {X 61.852,Y 94.791,Z 75.592,A 180.000,B 0.000,C 180.000} C_DIS
LIN {X 61.781,Y 94.757,Z 75.589,A 180.000,B 0.000,C 180.000} C_DIS
LIN {X 61.709,Y 94.725,Z 75.587,A 180.000,B 0.000,C 180.000} C_DIS
LIN {X 61.422,Y 94.596,Z 75.576,A 180.000,B 0.000,C 180.000} C_DIS
LIN {X 61.350,Y 94.564,Z 75.573,A 180.000,B 0.000,C 180.000} C_DIS
LIN {X 61.277,Y 94.533,Z 75.570,A 180.000,B 0.000,C 180.000} C_DIS
LIN {X 61.204,Y 94.505,Z 75.567,A 180.000,B 0.000,C 180.000} C_DIS
LIN {X 61.130,Y 94.479,Z 75.565,A 180.000,B 0.000,C 180.000} C_DIS
LIN {X 60.758,Y 94.350,Z 75.551,A 180.000,B 0.000,C 180.000} C_DIS
LIN {X 60.683,Y 94.325,Z 75.548,A 180.000,B 0.000,C 180.000} C_DIS
LIN {X 60.608,Y 94.302,Z 75.545,A 180.000,B 0.000,C 180.000} C_DIS
LIN {X 60.531,Y 94.282,Z 75.543,A 180.000,B 0.000,C 180.000} C_DIS
LIN {X 60.455,Y 94.263,Z 75.540,A 180.000,B 0.000,C 180.000} C_DIS
LIN {X 60.149,Y 94.187,Z 75.529,A 180.000,B 0.000,C 180.000} C_DIS
LIN {X 60.073,Y 94.168,Z 75.526,A 180.000,B 0.000,C 180.000} C_DIS
LIN {X 59.996,Y 94.151,Z 75.523,A 180.000,B 0.000,C 180.000} C_DIS
LIN {X 59.919,Y 94.136,Z 75.521,A 180.000,B 0.000,C 180.000} C_DIS
LIN {X 59.841,Y 94.123,Z 75.518,A 180.000,B 0.000,C 180.000} C_DIS
LIN {X 59.452,Y 94.063,Z 75.504,A 180.000,B 0.000,C 180.000} C_DIS
LIN {X 59.374,Y 94.051,Z 75.501,A 180.000,B 0.000,C 180.000} C_DIS
LIN {X 59.296,Y 94.042,Z 75.499,A 180.000,B 0.000,C 180.000} C_DIS
LIN {X 59.217,Y 94.036,Z 75.496,A 180.000,B 0.000,C 180.000} C_DIS
LIN {X 58.824,Y 94.010,Z 75.482,A 180.000,B 0.000,C 180.000} C_DIS
LIN {X 58.746,Y 94.005,Z 75.479,A 180.000,B 0.000,C 180.000} C_DIS
LIN {X 58.667,Y 94.002,Z 75.477,A 180.000,B 0.000,C 180.000} C_DIS
LIN {X 58.588,Y 94.001,Z 75.474,A 180.000,B 0.000,C 180.000} C_DIS
LIN {X 58.510,Y 94.003,Z 75.471,A 180.000,B 0.000,C 180.000} C_DIS
LIN {X 58.116,Y 94.012,Z 75.457,A 180.000,B 0.000,C 180.000} C_DIS
LIN {X 58.037,Y 94.014,Z 75.455,A 180.000,B 0.000,C 180.000} C_DIS
LIN {X 57.959,Y 94.020,Z 75.452,A 180.000,B 0.000,C 180.000} C_DIS
LIN {X 57.880,Y 94.028,Z 75.449,A 180.000,B 0.000,C 180.000} C_DIS
LIN {X 57.489,Y 94.071,Z 75.435,A 180.000,B 0.000,C 180.000} C_DIS
LIN {X 57.411,Y 94.080,Z 75.433,A 180.000,B 0.000,C 180.000} C_DIS
LIN {X 57.333,Y 94.091,Z 75.430,A 180.000,B 0.000,C 180.000} C_DIS
LIN {X 57.255,Y 94.105,Z 75.427,A 180.000,B 0.000,C 180.000} C_DIS
LIN {X 57.178,Y 94.121,Z 75.424,A 180.000,B 0.000,C 180.000} C_DIS
LIN {X 56.869,Y 94.183,Z 75.413,A 180.000,B 0.000,C 180.000} C_DIS
LIN {X 56.792,Y 94.199,Z 75.411,A 180.000,B 0.000,C 180.000} C_DIS
LIN {X 56.715,Y 94.216,Z 75.408,A 180.000,B 0.000,C 180.000} C_DIS
LIN {X 56.639,Y 94.235,Z 75.405,A 180.000,B 0.000,C 180.000} C_DIS
LIN {X 56.563,Y 94.257,Z 75.402,A 180.000,B 0.000,C 180.000} C_DIS
LIN {X 56.412,Y 94.301,Z 75.397,A 180.000,B 0.000,C 180.000} C_DIS
LIN {X 56.185,Y 94.368,Z 75.389,A 180.000,B 0.000,C 180.000} C_DIS
LIN {X 56.110,Y 94.391,Z 75.386,A 180.000,B 0.000,C 180.000} C_DIS
LIN {X 56.036,Y 94.417,Z 75.383,A 180.000,B 0.000,C 180.000} C_DIS
LIN {X 55.962,Y 94.444,Z 75.380,A 180.000,B 0.000,C 180.000} C_DIS
LIN {X 55.888,Y 94.473,Z 75.378,A 180.000,B 0.000,C 180.000} C_DIS
LIN {X 55.669,Y 94.560,Z 75.369,A 180.000,B 0.000,C 180.000} C_DIS
LIN {X 55.595,Y 94.589,Z 75.367,A 180.000,B 0.000,C 180.000} C_DIS
LIN {X 55.522,Y 94.618,Z 75.364,A 180.000,B 0.000,C 180.000} C_DIS
LIN {X 55.450,Y 94.648,Z 75.361,A 180.000,B 0.000,C 180.000} C_DIS
LIN {X 55.378,Y 94.681,Z 75.358,A 180.000,B 0.000,C 180.000} C_DIS
LIN {X 55.308,Y 94.716,Z 75.356,A 180.000,B 0.000,C 180.000} C_DIS
LIN {X 55.096,Y 94.822,Z 75.347,A 180.000,B 0.000,C 180.000} C_DIS
LIN {X 54.956,Y 94.893,Z 75.342,A 180.000,B 0.000,C 180.000} C_DIS
LIN {X 54.886,Y 94.929,Z 75.339,A 180.000,B 0.000,C 180.000} C_DIS
LIN {X 54.817,Y 94.967,Z 75.336,A 180.000,B 0.000,C 180.000} C_DIS
LIN {X 54.749,Y 95.007,Z 75.334,A 180.000,B 0.000,C 180.000} C_DIS
LIN {X 54.615,Y 95.090,Z 75.328,A 180.000,B 0.000,C 180.000} C_DIS
LIN {X 54.414,Y 95.214,Z 75.320,A 180.000,B 0.000,C 180.000} C_DIS
LIN {X 54.347,Y 95.256,Z 75.317,A 180.000,B 0.000,C 180.000} C_DIS
LIN {X 54.281,Y 95.299,Z 75.314,A 180.000,B 0.000,C 180.000} C_DIS
LIN {X 54.217,Y 95.344,Z 75.312,A 180.000,B 0.000,C 180.000} C_DIS
LIN {X 54.154,Y 95.391,Z 75.309,A 180.000,B 0.000,C 180.000} C_DIS
LIN {X 54.028,Y 95.486,Z 75.303,A 180.000,B 0.000,C 180.000} C_DIS
LIN {X 53.964,Y 95.533,Z 75.301,A 180.000,B 0.000,C 180.000} C_DIS
LIN {X 53.838,Y 95.627,Z 75.295,A 180.000,B 0.000,C 180.000} C_DIS
LIN {X 53.776,Y 95.675,Z 75.292,A 180.000,B 0.000,C 180.000} C_DIS
LIN {X 53.715,Y 95.725,Z 75.290,A 180.000,B 0.000,C 180.000} C_DIS
LIN {X 53.656,Y 95.777,Z 75.287,A 180.000,B 0.000,C 180.000} C_DIS
LIN {X 53.538,Y 95.882,Z 75.281,A 180.000,B 0.000,C 180.000} C_DIS
LIN {X 53.480,Y 95.935,Z 75.279,A 180.000,B 0.000,C 180.000} C_DIS
LIN {X 53.362,Y 96.040,Z 75.273,A 180.000,B 0.000,C 180.000} C_DIS
LIN {X 53.304,Y 96.092,Z 75.270,A 180.000,B 0.000,C 180.000} C_DIS
LIN {X 53.247,Y 96.147,Z 75.268,A 180.000,B 0.000,C 180.000} C_DIS
LIN {X 53.192,Y 96.203,Z 75.265,A 180.000,B 0.000,C 180.000} C_DIS
LIN {X 53.138,Y 96.260,Z 75.262,A 180.000,B 0.000,C 180.000} C_DIS
LIN {X 52.977,Y 96.433,Z 75.254,A 180.000,B 0.000,C 180.000} C_DIS
LIN {X 52.923,Y 96.490,Z 75.251,A 180.000,B 0.000,C 180.000} C_DIS
LIN {X 52.869,Y 96.548,Z 75.248,A 180.000,B 0.000,C 180.000} C_DIS
LIN {X 52.816,Y 96.607,Z 75.246,A 180.000,B 0.000,C 180.000} C_DIS
LIN {X 52.766,Y 96.667,Z 75.243,A 180.000,B 0.000,C 180.000} C_DIS
LIN {X 52.717,Y 96.728,Z 75.240,A 180.000,B 0.000,C 180.000} C_DIS
LIN {X 52.571,Y 96.915,Z 75.232,A 180.000,B 0.000,C 180.000} C_DIS
LIN {X 52.474,Y 97.039,Z 75.226,A 180.000,B 0.000,C 180.000} C_DIS
LIN {X 52.426,Y 97.101,Z 75.224,A 180.000,B 0.000,C 180.000} C_DIS
LIN {X 52.380,Y 97.165,Z 75.221,A 180.000,B 0.000,C 180.000} C_DIS
LIN {X 52.336,Y 97.230,Z 75.218,A 180.000,B 0.000,C 180.000} C_DIS
LIN {X 52.293,Y 97.296,Z 75.215,A 180.000,B 0.000,C 180.000} C_DIS
LIN {X 52.250,Y 97.362,Z 75.213,A 180.000,B 0.000,C 180.000} C_DIS
LIN {X 52.164,Y 97.494,Z 75.207,A 180.000,B 0.000,C 180.000} C_DIS
LIN {X 52.122,Y 97.561,Z 75.204,A 180.000,B 0.000,C 180.000} C_DIS
LIN {X 52.079,Y 97.627,Z 75.202,A 180.000,B 0.000,C 180.000} C_DIS
LIN {X 52.038,Y 97.694,Z 75.199,A 180.000,B 0.000,C 180.000} C_DIS
LIN {X 51.999,Y 97.762,Z 75.196,A 180.000,B 0.000,C 180.000} C_DIS
LIN {X 51.961,Y 97.832,Z 75.193,A 180.000,B 0.000,C 180.000} C_DIS
LIN {X 51.814,Y 98.110,Z 75.182,A 180.000,B 0.000,C 180.000} C_DIS
LIN {X 51.777,Y 98.180,Z 75.180,A 180.000,B 0.000,C 180.000} C_DIS
LIN {X 51.741,Y 98.250,Z 75.177,A 180.000,B 0.000,C 180.000} C_DIS
LIN {X 51.707,Y 98.321,Z 75.174,A 180.000,B 0.000,C 180.000} C_DIS
LIN {X 51.676,Y 98.393,Z 75.172,A 180.000,B 0.000,C 180.000} C_DIS
LIN {X 51.615,Y 98.538,Z 75.166,A 180.000,B 0.000,C 180.000} C_DIS
LIN {X 51.584,Y 98.611,Z 75.164,A 180.000,B 0.000,C 180.000} C_DIS
LIN {X 51.554,Y 98.683,Z 75.161,A 180.000,B 0.000,C 180.000} C_DIS
LIN {X 51.523,Y 98.756,Z 75.159,A 180.000,B 0.000,C 180.000} C_DIS
LIN {X 51.493,Y 98.829,Z 75.156,A 180.000,B 0.000,C 180.000} C_DIS
LIN {X 51.464,Y 98.902,Z 75.154,A 180.000,B 0.000,C 180.000} C_DIS
LIN {X 51.438,Y 98.976,Z 75.151,A 180.000,B 0.000,C 180.000} C_DIS
LIN {X 51.414,Y 99.051,Z 75.149,A 180.000,B 0.000,C 180.000} C_DIS
LIN {X 51.366,Y 99.201,Z 75.144,A 180.000,B 0.000,C 180.000} C_DIS
LIN {X 51.318,Y 99.351,Z 75.139,A 180.000,B 0.000,C 180.000} C_DIS
LIN {X 51.271,Y 99.502,Z 75.134,A 180.000,B 0.000,C 180.000} C_DIS
LIN {X 51.233,Y 99.654,Z 75.129,A 180.000,B 0.000,C 180.000} C_DIS
LIN {X 51.198,Y 99.808,Z 75.124,A 180.000,B 0.000,C 180.000} C_DIS
LIN {X 51.164,Y 99.962,Z 75.120,A 180.000,B 0.000,C 180.000} C_DIS
LIN {X 51.129,Y 100.115,Z 75.115,A 180.000,B 0.000,C 180.000} C_DIS
LIN {X 51.103,Y 100.271,Z 75.111,A 180.000,B 0.000,C 180.000} C_DIS
LIN {X 51.082,Y 100.427,Z 75.106,A 180.000,B 0.000,C 180.000} C_DIS
LIN {X 51.061,Y 100.583,Z 75.102,A 180.000,B 0.000,C 180.000} C_DIS
LIN {X 51.040,Y 100.739,Z 75.097,A 180.000,B 0.000,C 180.000} C_DIS
LIN {X 51.025,Y 100.896,Z 75.093,A 180.000,B 0.000,C 180.000} C_DIS
LIN {X 51.017,Y 101.053,Z 75.089,A 180.000,B 0.000,C 180.000} C_DIS
LIN {X 51.010,Y 101.210,Z 75.085,A 180.000,B 0.000,C 180.000} C_DIS
LIN {X 51.003,Y 101.368,Z 75.081,A 180.000,B 0.000,C 180.000} C_DIS
LIN {X 51.000,Y 101.525,Z 75.077,A 180.000,B 0.000,C 180.000} C_DIS
LIN {X 51.006,Y 101.683,Z 75.073,A 180.000,B 0.000,C 180.000} C_DIS
LIN {X 51.013,Y 101.840,Z 75.070,A 180.000,B 0.000,C 180.000} C_DIS
LIN {X 51.020,Y 101.997,Z 75.066,A 180.000,B 0.000,C 180.000} C_DIS
LIN {X 51.029,Y 102.155,Z 75.062,A 180.000,B 0.000,C 180.000} C_DIS
LIN {X 51.047,Y 102.311,Z 75.059,A 180.000,B 0.000,C 180.000} C_DIS
LIN {X 51.068,Y 102.467,Z 75.056,A 180.000,B 0.000,C 180.000} C_DIS
LIN {X 51.088,Y 102.623,Z 75.052,A 180.000,B 0.000,C 180.000} C_DIS
LIN {X 51.110,Y 102.779,Z 75.049,A 180.000,B 0.000,C 180.000} C_DIS
LIN {X 51.140,Y 102.934,Z 75.046,A 180.000,B 0.000,C 180.000} C_DIS
LIN {X 51.175,Y 103.087,Z 75.043,A 180.000,B 0.000,C 180.000} C_DIS
LIN {X 51.209,Y 103.241,Z 75.040,A 180.000,B 0.000,C 180.000} C_DIS
LIN {X 51.244,Y 103.395,Z 75.037,A 180.000,B 0.000,C 180.000} C_DIS
LIN {X 51.286,Y 103.547,Z 75.034,A 180.000,B 0.000,C 180.000} C_DIS
LIN {X 51.333,Y 103.697,Z 75.032,A 180.000,B 0.000,C 180.000} C_DIS
LIN {X 51.381,Y 103.847,Z 75.029,A 180.000,B 0.000,C 180.000} C_DIS
LIN {X 51.429,Y 103.997,Z 75.027,A 180.000,B 0.000,C 180.000} C_DIS
LIN {X 51.482,Y 104.145,Z 75.024,A 180.000,B 0.000,C 180.000} C_DIS
LIN {X 51.543,Y 104.291,Z 75.022,A 180.000,B 0.000,C 180.000} C_DIS
LIN {X 51.665,Y 104.581,Z 75.018,A 180.000,B 0.000,C 180.000} C_DIS
LIN {X 51.729,Y 104.725,Z 75.016,A 180.000,B 0.000,C 180.000} C_DIS
LIN {X 51.801,Y 104.865,Z 75.014,A 180.000,B 0.000,C 180.000} C_DIS
LIN {X 51.948,Y 105.143,Z 75.011,A 180.000,B 0.000,C 180.000} C_DIS
LIN {X 52.023,Y 105.282,Z 75.009,A 180.000,B 0.000,C 180.000} C_DIS
LIN {X 52.106,Y 105.416,Z 75.008,A 180.000,B 0.000,C 180.000} C_DIS
LIN {X 52.278,Y 105.680,Z 75.005,A 180.000,B 0.000,C 180.000} C_DIS
LIN {X 52.457,Y 105.939,Z 75.003,A 180.000,B 0.000,C 180.000} C_DIS
LIN {X 52.651,Y 106.187,Z 75.002,A 180.000,B 0.000,C 180.000} C_DIS
LIN {X 52.850,Y 106.431,Z 75.001,A 180.000,B 0.000,C 180.000} C_DIS
LIN {X 53.065,Y 106.661,Z 75.000,A 180.000,B 0.000,C 180.000} C_DIS
LIN {X 53.226,Y 106.829,Z 75.000,A 180.000,B 0.000,C 180.000} C_DIS
; Cutting Move Starts
LIN {X 53.277,Y 106.882,Z 75.000,A 180.000,B 0.000,C 180.000} C_DIS
LIN {X 53.304,Y 106.908,Z 75.000,A 180.000,B 0.000,C 180.000} C_DIS
LIN {X 53.455,Y 107.044,Z 75.000,A 180.000,B 0.000,C 180.000} C_DIS
LIN {X 53.634,Y 107.204,Z 75.000,A 180.000,B 0.000,C 180.000} C_DIS
LIN {X 53.704,Y 107.265,Z 75.000,A 180.000,B 0.000,C 180.000} C_DIS
LIN {X 53.813,Y 107.354,Z 75.000,A 180.000,B 0.000,C 180.000} C_DIS
LIN {X 53.933,Y 107.444,Z 75.000,A 180.000,B 0.000,C 180.000} C_DIS
LIN {X 54.172,Y 107.623,Z 75.000,A 180.000,B 0.000,C 180.000} C_DIS
LIN {X 54.349,Y 107.746,Z 75.000,A 180.000,B 0.000,C 180.000} C_DIS
LIN {X 54.439,Y 107.802,Z 75.000,A 180.000,B 0.000,C 180.000} C_DIS
LIN {X 54.729,Y 107.980,Z 75.000,A 180.000,B 0.000,C 180.000} C_DIS
LIN {X 54.886,Y 108.071,Z 75.000,A 180.000,B 0.000,C 180.000} C_DIS
LIN {X 55.059,Y 108.159,Z 75.000,A 180.000,B 0.000,C 180.000} C_DIS
LIN {X 55.243,Y 108.251,Z 75.000,A 180.000,B 0.000,C 180.000} C_DIS
LIN {X 55.419,Y 108.338,Z 75.000,A 180.000,B 0.000,C 180.000} C_DIS
LIN {X 55.422,Y 108.339,Z 75.000,A 180.000,B 0.000,C 180.000} C_DIS
LIN {X 55.601,Y 108.413,Z 75.000,A 180.000,B 0.000,C 180.000} C_DIS
LIN {X 55.862,Y 108.517,Z 75.000,A 180.000,B 0.000,C 180.000} C_DIS
LIN {X 55.958,Y 108.555,Z 75.000,A 180.000,B 0.000,C 180.000} C_DIS
LIN {X 56.137,Y 108.617,Z 75.000,A 180.000,B 0.000,C 180.000} C_DIS
LIN {X 56.316,Y 108.670,Z 75.000,A 180.000,B 0.000,C 180.000} C_DIS
LIN {X 56.495,Y 108.723,Z 75.000,A 180.000,B 0.000,C 180.000} C_DIS
LIN {X 56.673,Y 108.774,Z 75.000,A 180.000,B 0.000,C 180.000} C_DIS
LIN {X 56.852,Y 108.814,Z 75.000,A 180.000,B 0.000,C 180.000} C_DIS
LIN {X 57.210,Y 108.886,Z 75.000,A 180.000,B 0.000,C 180.000} C_DIS
LIN {X 57.388,Y 108.917,Z 75.000,A 180.000,B 0.000,C 180.000} C_DIS
LIN {X 57.567,Y 108.938,Z 75.000,A 180.000,B 0.000,C 180.000} C_DIS
LIN {X 57.746,Y 108.957,Z 75.000,A 180.000,B 0.000,C 180.000} C_DIS
LIN {X 57.925,Y 108.977,Z 75.000,A 180.000,B 0.000,C 180.000} C_DIS
LIN {X 58.103,Y 108.988,Z 75.000,A 180.000,B 0.000,C 180.000} C_DIS
LIN {X 58.282,Y 108.992,Z 75.000,A 180.000,B 0.000,C 180.000} C_DIS
LIN {X 58.461,Y 108.996,Z 75.000,A 180.000,B 0.000,C 180.000} C_DIS
LIN {X 58.640,Y 108.999,Z 75.000,A 180.000,B 0.000,C 180.000} C_DIS
LIN {X 58.819,Y 108.990,Z 75.000,A 180.000,B 0.000,C 180.000} C_DIS
LIN {X 59.176,Y 108.967,Z 75.000,A 180.000,B 0.000,C 180.000} C_DIS
LIN {X 59.355,Y 108.951,Z 75.000,A 180.000,B 0.000,C 180.000} C_DIS
LIN {X 59.534,Y 108.925,Z 75.000,A 180.000,B 0.000,C 180.000} C_DIS
LIN {X 59.856,Y 108.874,Z 75.000,A 180.000,B 0.000,C 180.000} C_DIS
LIN {X 59.891,Y 108.869,Z 75.000,A 180.000,B 0.000,C 180.000} C_DIS
LIN {X 60.070,Y 108.833,Z 75.000,A 180.000,B 0.000,C 180.000} C_DIS
LIN {X 60.249,Y 108.788,Z 75.000,A 180.000,B 0.000,C 180.000} C_DIS
LIN {X 60.427,Y 108.744,Z 75.000,A 180.000,B 0.000,C 180.000} C_DIS
LIN {X 60.606,Y 108.698,Z 75.000,A 180.000,B 0.000,C 180.000} C_DIS
LIN {X 60.616,Y 108.695,Z 75.000,A 180.000,B 0.000,C 180.000} C_DIS
LIN {X 60.785,Y 108.640,Z 75.000,A 180.000,B 0.000,C 180.000} C_DIS
LIN {X 61.144,Y 108.517,Z 75.000,A 180.000,B 0.000,C 180.000} C_DIS
LIN {X 61.321,Y 108.448,Z 75.000,A 180.000,B 0.000,C 180.000} C_DIS
LIN {X 61.500,Y 108.369,Z 75.000,A 180.000,B 0.000,C 180.000} C_DIS
LIN {X 61.679,Y 108.289,Z 75.000,A 180.000,B 0.000,C 180.000} C_DIS
LIN {X 61.858,Y 108.206,Z 75.000,A 180.000,B 0.000,C 180.000} C_DIS
LIN {X 61.948,Y 108.159,Z 75.000,A 180.000,B 0.000,C 180.000} C_DIS
LIN {X 62.036,Y 108.110,Z 75.000,A 180.000,B 0.000,C 180.000} C_DIS
LIN {X 62.268,Y 107.980,Z 75.000,A 180.000,B 0.000,C 180.000} C_DIS
LIN {X 62.394,Y 107.909,Z 75.000,A 180.000,B 0.000,C 180.000} C_DIS
LIN {X 62.562,Y 107.802,Z 75.000,A 180.000,B 0.000,C 180.000} C_DIS
LIN {X 62.825,Y 107.623,Z 75.000,A 180.000,B 0.000,C 180.000} C_DIS
LIN {X 62.930,Y 107.551,Z 75.000,A 180.000,B 0.000,C 180.000} C_DIS
LIN {X 63.071,Y 107.444,Z 75.000,A 180.000,B 0.000,C 180.000} C_DIS
LIN {X 63.109,Y 107.413,Z 75.000,A 180.000,B 0.000,C 180.000} C_DIS
LIN {X 63.290,Y 107.265,Z 75.000,A 180.000,B 0.000,C 180.000} C_DIS
LIN {X 63.467,Y 107.120,Z 75.000,A 180.000,B 0.000,C 180.000} C_DIS
LIN {X 63.504,Y 107.086,Z 75.000,A 180.000,B 0.000,C 180.000} C_DIS
LIN {X 63.645,Y 106.952,Z 75.000,A 180.000,B 0.000,C 180.000} C_DIS
LIN {X 63.873,Y 106.729,Z 75.000,A 180.000,B 0.000,C 180.000} C_DIS
LIN {X 64.003,Y 106.596,Z 75.000,A 180.000,B 0.000,C 180.000} C_DIS
LIN {X 64.043,Y 106.550,Z 75.000,A 180.000,B 0.000,C 180.000} C_DIS
LIN {X 64.196,Y 106.371,Z 75.000,A 180.000,B 0.000,C 180.000} C_DIS
LIN {X 64.349,Y 106.193,Z 75.000,A 180.000,B 0.000,C 180.000} C_DIS
LIN {X 64.360,Y 106.179,Z 75.000,A 180.000,B 0.000,C 180.000} C_DIS
LIN {X 64.487,Y 106.014,Z 75.000,A 180.000,B 0.000,C 180.000} C_DIS
LIN {X 64.718,Y 105.690,Z 75.000,A 180.000,B 0.000,C 180.000} C_DIS
LIN {X 64.742,Y 105.656,Z 75.000,A 180.000,B 0.000,C 180.000} C_DIS
LIN {X 64.856,Y 105.477,Z 75.000,A 180.000,B 0.000,C 180.000} C_DIS
LIN {X 65.075,Y 105.104,Z 75.000,A 180.000,B 0.000,C 180.000} C_DIS
LIN {X 65.163,Y 104.941,Z 75.000,A 180.000,B 0.000,C 180.000} C_DIS
LIN {X 65.248,Y 104.762,Z 75.000,A 180.000,B 0.000,C 180.000} C_DIS
LIN {X 65.333,Y 104.584,Z 75.000,A 180.000,B 0.000,C 180.000} C_DIS
LIN {X 65.415,Y 104.405,Z 75.000,A 180.000,B 0.000,C 180.000} C_DIS
LIN {X 65.433,Y 104.360,Z 75.000,A 180.000,B 0.000,C 180.000} C_DIS
LIN {X 65.483,Y 104.226,Z 75.000,A 180.000,B 0.000,C 180.000} C_DIS
LIN {X 65.549,Y 104.047,Z 75.000,A 180.000,B 0.000,C 180.000} C_DIS
LIN {X 65.612,Y 103.878,Z 75.000,A 180.000,B 0.000,C 180.000} C_DIS
LIN {X 65.615,Y 103.869,Z 75.000,A 180.000,B 0.000,C 180.000} C_DIS
LIN {X 65.672,Y 103.690,Z 75.000,A 180.000,B 0.000,C 180.000} C_DIS
LIN {X 65.720,Y 103.511,Z 75.000,A 180.000,B 0.000,C 180.000} C_DIS
LIN {X 65.791,Y 103.253,Z 75.000,A 180.000,B 0.000,C 180.000} C_DIS
LIN {X 65.815,Y 103.153,Z 75.000,A 180.000,B 0.000,C 180.000} C_DIS
LIN {X 65.850,Y 102.975,Z 75.000,A 180.000,B 0.000,C 180.000} C_DIS
LIN {X 65.914,Y 102.617,Z 75.000,A 180.000,B 0.000,C 180.000} C_DIS
LIN {X 65.941,Y 102.438,Z 75.000,A 180.000,B 0.000,C 180.000} C_DIS
LIN {X 65.957,Y 102.260,Z 75.000,A 180.000,B 0.000,C 180.000} C_DIS
LIN {X 65.973,Y 102.081,Z 75.000,A 180.000,B 0.000,C 180.000} C_DIS
LIN {X 65.989,Y 101.902,Z 75.000,A 180.000,B 0.000,C 180.000} C_DIS
LIN {X 65.995,Y 101.723,Z 75.000,A 180.000,B 0.000,C 180.000} C_DIS
LIN {X 65.995,Y 101.366,Z 75.000,A 180.000,B 0.000,C 180.000} C_DIS
LIN {X 65.993,Y 101.187,Z 75.000,A 180.000,B 0.000,C 180.000} C_DIS
LIN {X 65.981,Y 101.008,Z 75.000,A 180.000,B 0.000,C 180.000} C_DIS
LIN {X 65.949,Y 100.651,Z 75.000,A 180.000,B 0.000,C 180.000} C_DIS
LIN {X 65.929,Y 100.472,Z 75.000,A 180.000,B 0.000,C 180.000} C_DIS
LIN {X 65.898,Y 100.293,Z 75.000,A 180.000,B 0.000,C 180.000} C_DIS
LIN {X 65.866,Y 100.114,Z 75.000,A 180.000,B 0.000,C 180.000} C_DIS
LIN {X 65.834,Y 99.936,Z 75.000,A 180.000,B 0.000,C 180.000} C_DIS
LIN {X 65.793,Y 99.757,Z 75.000,A 180.000,B 0.000,C 180.000} C_DIS
LIN {X 65.791,Y 99.747,Z 75.000,A 180.000,B 0.000,C 180.000} C_DIS
LIN {X 65.696,Y 99.399,Z 75.000,A 180.000,B 0.000,C 180.000} C_DIS
LIN {X 65.645,Y 99.221,Z 75.000,A 180.000,B 0.000,C 180.000} C_DIS
LIN {X 65.612,Y 99.122,Z 75.000,A 180.000,B 0.000,C 180.000} C_DIS
LIN {X 65.582,Y 99.042,Z 75.000,A 180.000,B 0.000,C 180.000} C_DIS
LIN {X 65.516,Y 98.863,Z 75.000,A 180.000,B 0.000,C 180.000} C_DIS
LIN {X 65.450,Y 98.684,Z 75.000,A 180.000,B 0.000,C 180.000} C_DIS
LIN {X 65.433,Y 98.640,Z 75.000,A 180.000,B 0.000,C 180.000} C_DIS
LIN {X 65.375,Y 98.505,Z 75.000,A 180.000,B 0.000,C 180.000} C_DIS
LIN {X 65.290,Y 98.327,Z 75.000,A 180.000,B 0.000,C 180.000} C_DIS
LIN {X 65.206,Y 98.148,Z 75.000,A 180.000,B 0.000,C 180.000} C_DIS
LIN {X 65.117,Y 97.969,Z 75.000,A 180.000,B 0.000,C 180.000} C_DIS
LIN {X 65.075,Y 97.896,Z 75.000,A 180.000,B 0.000,C 180.000} C_DIS
LIN {X 64.897,Y 97.592,Z 75.000,A 180.000,B 0.000,C 180.000} C_DIS
LIN {X 64.801,Y 97.433,Z 75.000,A 180.000,B 0.000,C 180.000} C_DIS
LIN {X 64.718,Y 97.310,Z 75.000,A 180.000,B 0.000,C 180.000} C_DIS
LIN {X 64.539,Y 97.060,Z 75.000,A 180.000,B 0.000,C 180.000} C_DIS
LIN {X 64.421,Y 96.897,Z 75.000,A 180.000,B 0.000,C 180.000} C_DIS
LIN {X 64.360,Y 96.821,Z 75.000,A 180.000,B 0.000,C 180.000} C_DIS
LIN {X 64.272,Y 96.718,Z 75.000,A 180.000,B 0.000,C 180.000} C_DIS
LIN {X 64.119,Y 96.539,Z 75.000,A 180.000,B 0.000,C 180.000} C_DIS
LIN {X 64.003,Y 96.404,Z 75.000,A 180.000,B 0.000,C 180.000} C_DIS
LIN {X 63.962,Y 96.360,Z 75.000,A 180.000,B 0.000,C 180.000} C_DIS
LIN {X 63.824,Y 96.223,Z 75.000,A 180.000,B 0.000,C 180.000} C_DIS
LIN {X 63.599,Y 96.003,Z 75.000,A 180.000,B 0.000,C 180.000} C_DIS
LIN {X 63.467,Y 95.880,Z 75.000,A 180.000,B 0.000,C 180.000} C_DIS
LIN {X 63.399,Y 95.824,Z 75.000,A 180.000,B 0.000,C 180.000} C_DIS
LIN {X 63.109,Y 95.587,Z 75.000,A 180.000,B 0.000,C 180.000} C_DIS
LIN {X 62.954,Y 95.466,Z 75.000,A 180.000,B 0.000,C 180.000} C_DIS
LIN {X 62.930,Y 95.449,Z 75.000,A 180.000,B 0.000,C 180.000} C_DIS
LIN {X 62.751,Y 95.327,Z 75.000,A 180.000,B 0.000,C 180.000} C_DIS
LIN {X 62.573,Y 95.206,Z 75.000,A 180.000,B 0.000,C 180.000} C_DIS
LIN {X 62.425,Y 95.109,Z 75.000,A 180.000,B 0.000,C 180.000} C_DIS
LIN {X 62.394,Y 95.091,Z 75.000,A 180.000,B 0.000,C 180.000} C_DIS
LIN {X 62.215,Y 94.990,Z 75.000,A 180.000,B 0.000,C 180.000} C_DIS
LIN {X 62.036,Y 94.890,Z 75.000,A 180.000,B 0.000,C 180.000} C_DIS
LIN {X 61.858,Y 94.794,Z 75.000,A 180.000,B 0.000,C 180.000} C_DIS
LIN {X 61.769,Y 94.751,Z 75.000,A 180.000,B 0.000,C 180.000} C_DIS
LIN {X 61.679,Y 94.711,Z 75.000,A 180.000,B 0.000,C 180.000} C_DIS
LIN {X 61.369,Y 94.573,Z 75.000,A 180.000,B 0.000,C 180.000} C_DIS
LIN {X 61.321,Y 94.552,Z 75.000,A 180.000,B 0.000,C 180.000} C_DIS
LIN {X 61.143,Y 94.483,Z 75.000,A 180.000,B 0.000,C 180.000} C_DIS
LIN {X 60.785,Y 94.360,Z 75.000,A 180.000,B 0.000,C 180.000} C_DIS
LIN {X 60.606,Y 94.302,Z 75.000,A 180.000,B 0.000,C 180.000} C_DIS
LIN {X 60.427,Y 94.256,Z 75.000,A 180.000,B 0.000,C 180.000} C_DIS
LIN {X 60.249,Y 94.212,Z 75.000,A 180.000,B 0.000,C 180.000} C_DIS
LIN {X 60.070,Y 94.167,Z 75.000,A 180.000,B 0.000,C 180.000} C_DIS
LIN {X 59.891,Y 94.131,Z 75.000,A 180.000,B 0.000,C 180.000} C_DIS
LIN {X 59.712,Y 94.103,Z 75.000,A 180.000,B 0.000,C 180.000} C_DIS
LIN {X 59.534,Y 94.075,Z 75.000,A 180.000,B 0.000,C 180.000} C_DIS
LIN {X 59.355,Y 94.049,Z 75.000,A 180.000,B 0.000,C 180.000} C_DIS
LIN {X 59.220,Y 94.036,Z 75.000,A 180.000,B 0.000,C 180.000} C_DIS
LIN {X 58.819,Y 94.010,Z 75.000,A 180.000,B 0.000,C 180.000} C_DIS
LIN {X 58.640,Y 94.001,Z 75.000,A 180.000,B 0.000,C 180.000} C_DIS
LIN {X 58.461,Y 94.004,Z 75.000,A 180.000,B 0.000,C 180.000} C_DIS
LIN {X 58.282,Y 94.008,Z 75.000,A 180.000,B 0.000,C 180.000} C_DIS
LIN {X 58.103,Y 94.012,Z 75.000,A 180.000,B 0.000,C 180.000} C_DIS
LIN {X 57.925,Y 94.023,Z 75.000,A 180.000,B 0.000,C 180.000} C_DIS
LIN {X 57.803,Y 94.036,Z 75.000,A 180.000,B 0.000,C 180.000} C_DIS
LIN {X 57.567,Y 94.062,Z 75.000,A 180.000,B 0.000,C 180.000} C_DIS
LIN {X 57.388,Y 94.083,Z 75.000,A 180.000,B 0.000,C 180.000} C_DIS
LIN {X 57.210,Y 94.114,Z 75.000,A 180.000,B 0.000,C 180.000} C_DIS
LIN {X 56.852,Y 94.186,Z 75.000,A 180.000,B 0.000,C 180.000} C_DIS
LIN {X 56.717,Y 94.215,Z 75.000,A 180.000,B 0.000,C 180.000} C_DIS
LIN {X 56.673,Y 94.226,Z 75.000,A 180.000,B 0.000,C 180.000} C_DIS
LIN {X 56.495,Y 94.277,Z 75.000,A 180.000,B 0.000,C 180.000} C_DIS
LIN {X 56.316,Y 94.330,Z 75.000,A 180.000,B 0.000,C 180.000} C_DIS
LIN {X 56.137,Y 94.383,Z 75.000,A 180.000,B 0.000,C 180.000} C_DIS
LIN {X 56.103,Y 94.394,Z 75.000,A 180.000,B 0.000,C 180.000} C_DIS
LIN {X 55.958,Y 94.445,Z 75.000,A 180.000,B 0.000,C 180.000} C_DIS
LIN {X 55.601,Y 94.587,Z 75.000,A 180.000,B 0.000,C 180.000} C_DIS
LIN {X 55.422,Y 94.661,Z 75.000,A 180.000,B 0.000,C 180.000} C_DIS
LIN {X 55.243,Y 94.749,Z 75.000,A 180.000,B 0.000,C 180.000} C_DIS
LIN {X 55.064,Y 94.838,Z 75.000,A 180.000,B 0.000,C 180.000} C_DIS
LIN {X 54.886,Y 94.929,Z 75.000,A 180.000,B 0.000,C 180.000} C_DIS
LIN {X 54.883,Y 94.930,Z 75.000,A 180.000,B 0.000,C 180.000} C_DIS
LIN {X 54.707,Y 95.033,Z 75.000,A 180.000,B 0.000,C 180.000} C_DIS
LIN {X 54.528,Y 95.144,Z 75.000,A 180.000,B 0.000,C 180.000} C_DIS
LIN {X 54.349,Y 95.254,Z 75.000,A 180.000,B 0.000,C 180.000} C_DIS
LIN {X 54.298,Y 95.288,Z 75.000,A 180.000,B 0.000,C 180.000} C_DIS
LIN {X 54.171,Y 95.379,Z 75.000,A 180.000,B 0.000,C 180.000} C_DIS
LIN {X 53.992,Y 95.512,Z 75.000,A 180.000,B 0.000,C 180.000} C_DIS
LIN {X 53.814,Y 95.645,Z 75.000,A 180.000,B 0.000,C 180.000} C_DIS
LIN {X 53.813,Y 95.646,Z 75.000,A 180.000,B 0.000,C 180.000} C_DIS
LIN {X 53.634,Y 95.796,Z 75.000,A 180.000,B 0.000,C 180.000} C_DIS
LIN {X 53.404,Y 96.003,Z 75.000,A 180.000,B 0.000,C 180.000} C_DIS
LIN {X 53.277,Y 96.118,Z 75.000,A 180.000,B 0.000,C 180.000} C_DIS
LIN {X 53.213,Y 96.181,Z 75.000,A 180.000,B 0.000,C 180.000} C_DIS
LIN {X 53.098,Y 96.303,Z 75.000,A 180.000,B 0.000,C 180.000} C_DIS
LIN {X 52.877,Y 96.539,Z 75.000,A 180.000,B 0.000,C 180.000} C_DIS
LIN {X 52.740,Y 96.698,Z 75.000,A 180.000,B 0.000,C 180.000} C_DIS
LIN {X 52.725,Y 96.718,Z 75.000,A 180.000,B 0.000,C 180.000} C_DIS
LIN {X 52.562,Y 96.927,Z 75.000,A 180.000,B 0.000,C 180.000} C_DIS
LIN {X 52.446,Y 97.075,Z 75.000,A 180.000,B 0.000,C 180.000} C_DIS
LIN {X 52.383,Y 97.161,Z 75.000,A 180.000,B 0.000,C 180.000} C_DIS
LIN {X 52.320,Y 97.254,Z 75.000,A 180.000,B 0.000,C 180.000} C_DIS
LIN {X 52.088,Y 97.612,Z 75.000,A 180.000,B 0.000,C 180.000} C_DIS
LIN {X 52.025,Y 97.715,Z 75.000,A 180.000,B 0.000,C 180.000} C_DIS
LIN {X 51.983,Y 97.790,Z 75.000,A 180.000,B 0.000,C 180.000} C_DIS
LIN {X 51.889,Y 97.969,Z 75.000,A 180.000,B 0.000,C 180.000} C_DIS
LIN {X 51.794,Y 98.148,Z 75.000,A 180.000,B 0.000,C 180.000} C_DIS
LIN {X 51.705,Y 98.327,Z 75.000,A 180.000,B 0.000,C 180.000} C_DIS
LIN {X 51.668,Y 98.412,Z 75.000,A 180.000,B 0.000,C 180.000} C_DIS
LIN {X 51.553,Y 98.684,Z 75.000,A 180.000,B 0.000,C 180.000} C_DIS
LIN {X 51.489,Y 98.838,Z 75.000,A 180.000,B 0.000,C 180.000} C_DIS
LIN {X 51.479,Y 98.863,Z 75.000,A 180.000,B 0.000,C 180.000} C_DIS
LIN {X 51.417,Y 99.042,Z 75.000,A 180.000,B 0.000,C 180.000} C_DIS
LIN {X 51.303,Y 99.399,Z 75.000,A 180.000,B 0.000,C 180.000} C_DIS
LIN {X 51.251,Y 99.578,Z 75.000,A 180.000,B 0.000,C 180.000} C_DIS
LIN {X 51.210,Y 99.757,Z 75.000,A 180.000,B 0.000,C 180.000} C_DIS
LIN {X 51.170,Y 99.936,Z 75.000,A 180.000,B 0.000,C 180.000} C_DIS
LIN {X 51.131,Y 100.106,Z 75.000,A 180.000,B 0.000,C 180.000} C_DIS
LIN {X 51.130,Y 100.114,Z 75.000,A 180.000,B 0.000,C 180.000} C_DIS
LIN {X 51.100,Y 100.293,Z 75.000,A 180.000,B 0.000,C 180.000} C_DIS
LIN {X 51.052,Y 100.651,Z 75.000,A 180.000,B 0.000,C 180.000} C_DIS
LIN {X 51.030,Y 100.829,Z 75.000,A 180.000,B 0.000,C 180.000} C_DIS
LIN {X 51.019,Y 101.008,Z 75.000,A 180.000,B 0.000,C 180.000} C_DIS
LIN {X 51.003,Y 101.366,Z 75.000,A 180.000,B 0.000,C 180.000} C_DIS
LIN {X 51.000,Y 101.545,Z 75.000,A 180.000,B 0.000,C 180.000} C_DIS
LIN {X 51.007,Y 101.723,Z 75.000,A 180.000,B 0.000,C 180.000} C_DIS
LIN {X 51.015,Y 101.902,Z 75.000,A 180.000,B 0.000,C 180.000} C_DIS
LIN {X 51.023,Y 102.081,Z 75.000,A 180.000,B 0.000,C 180.000} C_DIS
LIN {X 51.040,Y 102.260,Z 75.000,A 180.000,B 0.000,C 180.000} C_DIS
LIN {X 51.064,Y 102.438,Z 75.000,A 180.000,B 0.000,C 180.000} C_DIS
LIN {X 51.088,Y 102.617,Z 75.000,A 180.000,B 0.000,C 180.000} C_DIS
LIN {X 51.113,Y 102.796,Z 75.000,A 180.000,B 0.000,C 180.000} C_DIS
LIN {X 51.131,Y 102.894,Z 75.000,A 180.000,B 0.000,C 180.000} C_DIS
LIN {X 51.149,Y 102.975,Z 75.000,A 180.000,B 0.000,C 180.000} C_DIS
LIN {X 51.230,Y 103.332,Z 75.000,A 180.000,B 0.000,C 180.000} C_DIS
LIN {X 51.275,Y 103.511,Z 75.000,A 180.000,B 0.000,C 180.000} C_DIS
LIN {X 51.310,Y 103.624,Z 75.000,A 180.000,B 0.000,C 180.000} C_DIS
LIN {X 51.388,Y 103.869,Z 75.000,A 180.000,B 0.000,C 180.000} C_DIS
LIN {X 51.446,Y 104.047,Z 75.000,A 180.000,B 0.000,C 180.000} C_DIS
LIN {X 51.489,Y 104.162,Z 75.000,A 180.000,B 0.000,C 180.000} C_DIS
LIN {X 51.515,Y 104.226,Z 75.000,A 180.000,B 0.000,C 180.000} C_DIS
LIN {X 51.668,Y 104.588,Z 75.000,A 180.000,B 0.000,C 180.000} C_DIS
LIN {X 51.747,Y 104.762,Z 75.000,A 180.000,B 0.000,C 180.000} C_DIS
LIN {X 51.841,Y 104.941,Z 75.000,A 180.000,B 0.000,C 180.000} C_DIS
LIN {X 51.936,Y 105.120,Z 75.000,A 180.000,B 0.000,C 180.000} C_DIS
LIN {X 52.025,Y 105.285,Z 75.000,A 180.000,B 0.000,C 180.000} C_DIS
LIN {X 52.033,Y 105.299,Z 75.000,A 180.000,B 0.000,C 180.000} C_DIS
LIN {X 52.146,Y 105.477,Z 75.000,A 180.000,B 0.000,C 180.000} C_DIS
LIN {X 52.262,Y 105.656,Z 75.000,A 180.000,B 0.000,C 180.000} C_DIS
LIN {X 52.380,Y 105.835,Z 75.000,A 180.000,B 0.000,C 180.000} C_DIS
LIN {X 52.383,Y 105.839,Z 75.000,A 180.000,B 0.000,C 180.000} C_DIS
LIN {X 52.515,Y 106.014,Z 75.000,A 180.000,B 0.000,C 180.000} C_DIS
LIN {X 52.655,Y 106.193,Z 75.000,A 180.000,B 0.000,C 180.000} C_DIS
LIN {X 52.740,Y 106.302,Z 75.000,A 180.000,B 0.000,C 180.000} C_DIS
LIN {X 52.797,Y 106.371,Z 75.000,A 180.000,B 0.000,C 180.000} C_DIS
LIN {X 52.919,Y 106.506,Z 75.000,A 180.000,B 0.000,C 180.000} C_DIS
LIN {X 53.128,Y 106.729,Z 75.000,A 180.000,B 0.000,C 180.000} C_DIS
LIN {X 53.226,Y 106.829,Z 75.000,A 180.000,B 0.000,C 180.000} C_DIS
; Link Move Starts
LIN {X 53.456,Y 107.044,Z 75.000,A 180.000,B 0.000,C 180.000} C_DIS
LIN {X 53.691,Y 107.254,Z 74.998,A 180.000,B 0.000,C 180.000} C_DIS
LIN {X 53.939,Y 107.448,Z 74.996,A 180.000,B 0.000,C 180.000} C_DIS
LIN {X 54.191,Y 107.637,Z 74.992,A 180.000,B 0.000,C 180.000} C_DIS
LIN {X 54.320,Y 107.727,Z 74.991,A 180.000,B 0.000,C 180.000} C_DIS
LIN {X 54.454,Y 107.810,Z 74.988,A 180.000,B 0.000,C 180.000} C_DIS
LIN {X 54.722,Y 107.976,Z 74.983,A 180.000,B 0.000,C 180.000} C_DIS
LIN {X 54.858,Y 108.056,Z 74.981,A 180.000,B 0.000,C 180.000} C_DIS
LIN {X 54.998,Y 108.128,Z 74.978,A 180.000,B 0.000,C 180.000} C_DIS
LIN {X 55.138,Y 108.199,Z 74.975,A 180.000,B 0.000,C 180.000} C_DIS
LIN {X 55.279,Y 108.270,Z 74.971,A 180.000,B 0.000,C 180.000} C_DIS
LIN {X 55.421,Y 108.339,Z 74.968,A 180.000,B 0.000,C 180.000} C_DIS
LIN {X 55.566,Y 108.400,Z 74.964,A 180.000,B 0.000,C 180.000} C_DIS
LIN {X 55.712,Y 108.458,Z 74.960,A 180.000,B 0.000,C 180.000} C_DIS
LIN {X 55.859,Y 108.515,Z 74.956,A 180.000,B 0.000,C 180.000} C_DIS
LIN {X 56.006,Y 108.573,Z 74.952,A 180.000,B 0.000,C 180.000} C_DIS
LIN {X 56.155,Y 108.622,Z 74.948,A 180.000,B 0.000,C 180.000} C_DIS
LIN {X 56.306,Y 108.667,Z 74.944,A 180.000,B 0.000,C 180.000} C_DIS
LIN {X 56.457,Y 108.712,Z 74.939,A 180.000,B 0.000,C 180.000} C_DIS
LIN {X 56.608,Y 108.756,Z 74.934,A 180.000,B 0.000,C 180.000} C_DIS
LIN {X 56.761,Y 108.795,Z 74.929,A 180.000,B 0.000,C 180.000} C_DIS
LIN {X 56.915,Y 108.826,Z 74.924,A 180.000,B 0.000,C 180.000} C_DIS
LIN {X 56.992,Y 108.842,Z 74.922,A 180.000,B 0.000,C 180.000} C_DIS
LIN {X 57.070,Y 108.858,Z 74.919,A 180.000,B 0.000,C 180.000} C_DIS
LIN {X 57.147,Y 108.873,Z 74.917,A 180.000,B 0.000,C 180.000} C_DIS
LIN {X 57.224,Y 108.889,Z 74.914,A 180.000,B 0.000,C 180.000} C_DIS
LIN {X 57.301,Y 108.903,Z 74.911,A 180.000,B 0.000,C 180.000} C_DIS
LIN {X 57.379,Y 108.916,Z 74.909,A 180.000,B 0.000,C 180.000} C_DIS
LIN {X 57.457,Y 108.925,Z 74.906,A 180.000,B 0.000,C 180.000} C_DIS
LIN {X 57.536,Y 108.934,Z 74.903,A 180.000,B 0.000,C 180.000} C_DIS
LIN {X 57.614,Y 108.943,Z 74.901,A 180.000,B 0.000,C 180.000} C_DIS
LIN {X 57.692,Y 108.951,Z 74.898,A 180.000,B 0.000,C 180.000} C_DIS
LIN {X 57.770,Y 108.960,Z 74.895,A 180.000,B 0.000,C 180.000} C_DIS
LIN {X 57.849,Y 108.969,Z 74.892,A 180.000,B 0.000,C 180.000} C_DIS
LIN {X 57.927,Y 108.977,Z 74.890,A 180.000,B 0.000,C 180.000} C_DIS
LIN {X 58.005,Y 108.984,Z 74.887,A 180.000,B 0.000,C 180.000} C_DIS
LIN {X 58.084,Y 108.988,Z 74.884,A 180.000,B 0.000,C 180.000} C_DIS
LIN {X 58.163,Y 108.989,Z 74.881,A 180.000,B 0.000,C 180.000} C_DIS
LIN {X 58.242,Y 108.991,Z 74.878,A 180.000,B 0.000,C 180.000} C_DIS
LIN {X 58.320,Y 108.993,Z 74.876,A 180.000,B 0.000,C 180.000} C_DIS
LIN {X 58.399,Y 108.995,Z 74.873,A 180.000,B 0.000,C 180.000} C_DIS
LIN {X 58.478,Y 108.996,Z 74.870,A 180.000,B 0.000,C 180.000} C_DIS
LIN {X 58.556,Y 108.998,Z 74.867,A 180.000,B 0.000,C 180.000} C_DIS
LIN {X 58.635,Y 108.999,Z 74.865,A 180.000,B 0.000,C 180.000} C_DIS
LIN {X 58.714,Y 108.997,Z 74.862,A 180.000,B 0.000,C 180.000} C_DIS
LIN {X 58.793,Y 108.992,Z 74.859,A 180.000,B 0.000,C 180.000} C_DIS
LIN {X 59.028,Y 108.977,Z 74.851,A 180.000,B 0.000,C 180.000} C_DIS
LIN {X 59.185,Y 108.966,Z 74.845,A 180.000,B 0.000,C 180.000} C_DIS
LIN {X 59.264,Y 108.960,Z 74.843,A 180.000,B 0.000,C 180.000} C_DIS
LIN {X 59.342,Y 108.953,Z 74.840,A 180.000,B 0.000,C 180.000} C_DIS
LIN {X 59.420,Y 108.942,Z 74.837,A 180.000,B 0.000,C 180.000} C_DIS
LIN {X 59.498,Y 108.930,Z 74.834,A 180.000,B 0.000,C 180.000} C_DIS
LIN {X 59.576,Y 108.918,Z 74.832,A 180.000,B 0.000,C 180.000} C_DIS
LIN {X 59.732,Y 108.894,Z 74.826,A 180.000,B 0.000,C 180.000} C_DIS
LIN {X 59.809,Y 108.881,Z 74.823,A 180.000,B 0.000,C 180.000} C_DIS
LIN {X 59.887,Y 108.869,Z 74.821,A 180.000,B 0.000,C 180.000} C_DIS
LIN {X 59.965,Y 108.856,Z 74.818,A 180.000,B 0.000,C 180.000} C_DIS
LIN {X 60.042,Y 108.839,Z 74.815,A 180.000,B 0.000,C 180.000} C_DIS
LIN {X 60.118,Y 108.821,Z 74.812,A 180.000,B 0.000,C 180.000} C_DIS
LIN {X 60.195,Y 108.802,Z 74.810,A 180.000,B 0.000,C 180.000} C_DIS
LIN {X 60.348,Y 108.764,Z 74.804,A 180.000,B 0.000,C 180.000} C_DIS
LIN {X 60.501,Y 108.726,Z 74.799,A 180.000,B 0.000,C 180.000} C_DIS
LIN {X 60.577,Y 108.706,Z 74.796,A 180.000,B 0.000,C 180.000} C_DIS
LIN {X 60.653,Y 108.684,Z 74.793,A 180.000,B 0.000,C 180.000} C_DIS
LIN {X 60.727,Y 108.660,Z 74.790,A 180.000,B 0.000,C 180.000} C_DIS
LIN {X 60.876,Y 108.609,Z 74.785,A 180.000,B 0.000,C 180.000} C_DIS
LIN {X 61.100,Y 108.532,Z 74.777,A 180.000,B 0.000,C 180.000} C_DIS
LIN {X 61.174,Y 108.506,Z 74.774,A 180.000,B 0.000,C 180.000} C_DIS
LIN {X 61.248,Y 108.478,Z 74.771,A 180.000,B 0.000,C 180.000} C_DIS
LIN {X 61.321,Y 108.449,Z 74.768,A 180.000,B 0.000,C 180.000} C_DIS
LIN {X 61.393,Y 108.417,Z 74.766,A 180.000,B 0.000,C 180.000} C_DIS
LIN {X 61.752,Y 108.256,Z 74.752,A 180.000,B 0.000,C 180.000} C_DIS
LIN {X 61.824,Y 108.223,Z 74.749,A 180.000,B 0.000,C 180.000} C_DIS
LIN {X 61.894,Y 108.188,Z 74.746,A 180.000,B 0.000,C 180.000} C_DIS
LIN {X 61.964,Y 108.150,Z 74.744,A 180.000,B 0.000,C 180.000} C_DIS
LIN {X 62.307,Y 107.959,Z 74.730,A 180.000,B 0.000,C 180.000} C_DIS
LIN {X 62.376,Y 107.920,Z 74.727,A 180.000,B 0.000,C 180.000} C_DIS
LIN {X 62.444,Y 107.879,Z 74.724,A 180.000,B 0.000,C 180.000} C_DIS
LIN {X 62.510,Y 107.837,Z 74.722,A 180.000,B 0.000,C 180.000} C_DIS
LIN {X 62.575,Y 107.793,Z 74.719,A 180.000,B 0.000,C 180.000} C_DIS
LIN {X 62.901,Y 107.571,Z 74.705,A 180.000,B 0.000,C 180.000} C_DIS
LIN {X 62.965,Y 107.526,Z 74.702,A 180.000,B 0.000,C 180.000} C_DIS
LIN {X 63.028,Y 107.479,Z 74.700,A 180.000,B 0.000,C 180.000} C_DIS
LIN {X 63.089,Y 107.429,Z 74.697,A 180.000,B 0.000,C 180.000} C_DIS
LIN {X 63.211,Y 107.329,Z 74.691,A 180.000,B 0.000,C 180.000} C_DIS
LIN {X 63.272,Y 107.280,Z 74.689,A 180.000,B 0.000,C 180.000} C_DIS
LIN {X 63.394,Y 107.180,Z 74.683,A 180.000,B 0.000,C 180.000} C_DIS
LIN {X 63.455,Y 107.130,Z 74.680,A 180.000,B 0.000,C 180.000} C_DIS
LIN {X 63.514,Y 107.078,Z 74.678,A 180.000,B 0.000,C 180.000} C_DIS
LIN {X 63.571,Y 107.024,Z 74.675,A 180.000,B 0.000,C 180.000} C_DIS
LIN {X 63.628,Y 106.969,Z 74.672,A 180.000,B 0.000,C 180.000} C_DIS
LIN {X 63.797,Y 106.804,Z 74.664,A 180.000,B 0.000,C 180.000} C_DIS
LIN {X 63.853,Y 106.749,Z 74.661,A 180.000,B 0.000,C 180.000} C_DIS
LIN {X 63.909,Y 106.693,Z 74.658,A 180.000,B 0.000,C 180.000} C_DIS
LIN {X 63.964,Y 106.637,Z 74.656,A 180.000,B 0.000,C 180.000} C_DIS
LIN {X 64.018,Y 106.579,Z 74.653,A 180.000,B 0.000,C 180.000} C_DIS
LIN {X 64.069,Y 106.520,Z 74.650,A 180.000,B 0.000,C 180.000} C_DIS
LIN {X 64.172,Y 106.400,Z 74.645,A 180.000,B 0.000,C 180.000} C_DIS
LIN {X 64.274,Y 106.280,Z 74.639,A 180.000,B 0.000,C 180.000} C_DIS
LIN {X 64.325,Y 106.221,Z 74.636,A 180.000,B 0.000,C 180.000} C_DIS
LIN {X 64.376,Y 106.160,Z 74.634,A 180.000,B 0.000,C 180.000} C_DIS
LIN {X 64.425,Y 106.098,Z 74.631,A 180.000,B 0.000,C 180.000} C_DIS
LIN {X 64.472,Y 106.035,Z 74.628,A 180.000,B 0.000,C 180.000} C_DIS
LIN {X 64.517,Y 105.971,Z 74.625,A 180.000,B 0.000,C 180.000} C_DIS
LIN {X 64.563,Y 105.907,Z 74.623,A 180.000,B 0.000,C 180.000} C_DIS
LIN {X 64.609,Y 105.843,Z 74.620,A 180.000,B 0.000,C 180.000} C_DIS
LIN {X 64.654,Y 105.779,Z 74.617,A 180.000,B 0.000,C 180.000} C_DIS
LIN {X 64.700,Y 105.715,Z 74.614,A 180.000,B 0.000,C 180.000} C_DIS
LIN {X 64.746,Y 105.650,Z 74.612,A 180.000,B 0.000,C 180.000} C_DIS
LIN {X 64.790,Y 105.585,Z 74.609,A 180.000,B 0.000,C 180.000} C_DIS
LIN {X 64.832,Y 105.518,Z 74.606,A 180.000,B 0.000,C 180.000} C_DIS
LIN {X 64.872,Y 105.451,Z 74.603,A 180.000,B 0.000,C 180.000} C_DIS
LIN {X 64.912,Y 105.383,Z 74.601,A 180.000,B 0.000,C 180.000} C_DIS
LIN {X 64.952,Y 105.315,Z 74.598,A 180.000,B 0.000,C 180.000} C_DIS
LIN {X 64.992,Y 105.247,Z 74.595,A 180.000,B 0.000,C 180.000} C_DIS
LIN {X 65.031,Y 105.179,Z 74.592,A 180.000,B 0.000,C 180.000} C_DIS
LIN {X 65.071,Y 105.111,Z 74.590,A 180.000,B 0.000,C 180.000} C_DIS
LIN {X 65.110,Y 105.043,Z 74.587,A 180.000,B 0.000,C 180.000} C_DIS
LIN {X 65.147,Y 104.973,Z 74.584,A 180.000,B 0.000,C 180.000} C_DIS
LIN {X 65.182,Y 104.902,Z 74.582,A 180.000,B 0.000,C 180.000} C_DIS
LIN {X 65.216,Y 104.831,Z 74.579,A 180.000,B 0.000,C 180.000} C_DIS
LIN {X 65.249,Y 104.760,Z 74.577,A 180.000,B 0.000,C 180.000} C_DIS
LIN {X 65.283,Y 104.689,Z 74.574,A 180.000,B 0.000,C 180.000} C_DIS
LIN {X 65.350,Y 104.546,Z 74.569,A 180.000,B 0.000,C 180.000} C_DIS
LIN {X 65.415,Y 104.403,Z 74.564,A 180.000,B 0.000,C 180.000} C_DIS
LIN {X 65.472,Y 104.256,Z 74.560,A 180.000,B 0.000,C 180.000} C_DIS
LIN {X 65.527,Y 104.108,Z 74.555,A 180.000,B 0.000,C 180.000} C_DIS
LIN {X 65.581,Y 103.961,Z 74.551,A 180.000,B 0.000,C 180.000} C_DIS
LIN {X 65.635,Y 103.812,Z 74.547,A 180.000,B 0.000,C 180.000} C_DIS
LIN {X 65.680,Y 103.661,Z 74.542,A 180.000,B 0.000,C 180.000} C_DIS
LIN {X 65.721,Y 103.509,Z 74.539,A 180.000,B 0.000,C 180.000} C_DIS
LIN {X 65.762,Y 103.357,Z 74.535,A 180.000,B 0.000,C 180.000} C_DIS
LIN {X 65.803,Y 103.205,Z 74.531,A 180.000,B 0.000,C 180.000} C_DIS
LIN {X 65.837,Y 103.051,Z 74.528,A 180.000,B 0.000,C 180.000} C_DIS
LIN {X 65.864,Y 102.896,Z 74.524,A 180.000,B 0.000,C 180.000} C_DIS
LIN {X 65.892,Y 102.741,Z 74.521,A 180.000,B 0.000,C 180.000} C_DIS
LIN {X 65.920,Y 102.586,Z 74.519,A 180.000,B 0.000,C 180.000} C_DIS
LIN {X 65.942,Y 102.430,Z 74.516,A 180.000,B 0.000,C 180.000} C_DIS
LIN {X 65.970,Y 102.117,Z 74.511,A 180.000,B 0.000,C 180.000} C_DIS
LIN {X 65.994,Y 101.803,Z 74.507,A 180.000,B 0.000,C 180.000} C_DIS
LIN {X 65.995,Y 101.488,Z 74.504,A 180.000,B 0.000,C 180.000} C_DIS
LIN {X 65.993,Y 101.173,Z 74.502,A 180.000,B 0.000,C 180.000} C_DIS
LIN {X 65.968,Y 100.859,Z 74.500,A 180.000,B 0.000,C 180.000} C_DIS
LIN {X 65.942,Y 100.588,Z 74.500,A 180.000,B 0.000,C 180.000} C_DIS
; Cutting Move Starts
LIN {X 65.929,Y 100.472,Z 74.500,A 180.000,B 0.000,C 180.000} C_DIS
LIN {X 65.898,Y 100.293,Z 74.500,A 180.000,B 0.000,C 180.000} C_DIS
LIN {X 65.866,Y 100.114,Z 74.500,A 180.000,B 0.000,C 180.000} C_DIS
LIN {X 65.834,Y 99.936,Z 74.500,A 180.000,B 0.000,C 180.000} C_DIS
LIN {X 65.793,Y 99.757,Z 74.500,A 180.000,B 0.000,C 180.000} C_DIS
LIN {X 65.791,Y 99.747,Z 74.500,A 180.000,B 0.000,C 180.000} C_DIS
LIN {X 65.696,Y 99.399,Z 74.500,A 180.000,B 0.000,C 180.000} C_DIS
LIN {X 65.645,Y 99.221,Z 74.500,A 180.000,B 0.000,C 180.000} C_DIS
LIN {X 65.612,Y 99.122,Z 74.500,A 180.000,B 0.000,C 180.000} C_DIS
LIN {X 65.582,Y 99.042,Z 74.500,A 180.000,B 0.000,C 180.000} C_DIS
LIN {X 65.516,Y 98.863,Z 74.500,A 180.000,B 0.000,C 180.000} C_DIS
LIN {X 65.450,Y 98.684,Z 74.500,A 180.000,B 0.000,C 180.000} C_DIS
LIN {X 65.433,Y 98.640,Z 74.500,A 180.000,B 0.000,C 180.000} C_DIS
LIN {X 65.375,Y 98.505,Z 74.500,A 180.000,B 0.000,C 180.000} C_DIS
LIN {X 65.290,Y 98.327,Z 74.500,A 180.000,B 0.000,C 180.000} C_DIS
LIN {X 65.206,Y 98.148,Z 74.500,A 180.000,B 0.000,C 180.000} C_DIS
LIN {X 65.117,Y 97.969,Z 74.500,A 180.000,B 0.000,C 180.000} C_DIS
LIN {X 65.075,Y 97.896,Z 74.500,A 180.000,B 0.000,C 180.000} C_DIS
LIN {X 64.897,Y 97.592,Z 74.500,A 180.000,B 0.000,C 180.000} C_DIS
LIN {X 64.801,Y 97.433,Z 74.500,A 180.000,B 0.000,C 180.000} C_DIS
LIN {X 64.718,Y 97.310,Z 74.500,A 180.000,B 0.000,C 180.000} C_DIS
LIN {X 64.539,Y 97.060,Z 74.500,A 180.000,B 0.000,C 180.000} C_DIS
LIN {X 64.421,Y 96.897,Z 74.500,A 180.000,B 0.000,C 180.000} C_DIS
LIN {X 64.360,Y 96.821,Z 74.500,A 180.000,B 0.000,C 180.000} C_DIS
LIN {X 64.272,Y 96.718,Z 74.500,A 180.000,B 0.000,C 180.000} C_DIS
LIN {X 64.119,Y 96.539,Z 74.500,A 180.000,B 0.000,C 180.000} C_DIS
LIN {X 64.003,Y 96.404,Z 74.500,A 180.000,B 0.000,C 180.000} C_DIS
LIN {X 63.962,Y 96.360,Z 74.500,A 180.000,B 0.000,C 180.000} C_DIS
LIN {X 63.824,Y 96.223,Z 74.500,A 180.000,B 0.000,C 180.000} C_DIS
LIN {X 63.599,Y 96.003,Z 74.500,A 180.000,B 0.000,C 180.000} C_DIS
LIN {X 63.467,Y 95.880,Z 74.500,A 180.000,B 0.000,C 180.000} C_DIS
LIN {X 63.399,Y 95.824,Z 74.500,A 180.000,B 0.000,C 180.000} C_DIS
LIN {X 63.109,Y 95.587,Z 74.500,A 180.000,B 0.000,C 180.000} C_DIS
LIN {X 62.954,Y 95.466,Z 74.500,A 180.000,B 0.000,C 180.000} C_DIS
LIN {X 62.930,Y 95.449,Z 74.500,A 180.000,B 0.000,C 180.000} C_DIS
LIN {X 62.751,Y 95.327,Z 74.500,A 180.000,B 0.000,C 180.000} C_DIS
LIN {X 62.573,Y 95.206,Z 74.500,A 180.000,B 0.000,C 180.000} C_DIS
LIN {X 62.425,Y 95.109,Z 74.500,A 180.000,B 0.000,C 180.000} C_DIS
LIN {X 62.394,Y 95.091,Z 74.500,A 180.000,B 0.000,C 180.000} C_DIS
LIN {X 62.215,Y 94.990,Z 74.500,A 180.000,B 0.000,C 180.000} C_DIS
LIN {X 62.036,Y 94.890,Z 74.500,A 180.000,B 0.000,C 180.000} C_DIS
LIN {X 61.858,Y 94.794,Z 74.500,A 180.000,B 0.000,C 180.000} C_DIS
LIN {X 61.769,Y 94.751,Z 74.500,A 180.000,B 0.000,C 180.000} C_DIS
LIN {X 61.679,Y 94.711,Z 74.500,A 180.000,B 0.000,C 180.000} C_DIS
LIN {X 61.369,Y 94.573,Z 74.500,A 180.000,B 0.000,C 180.000} C_DIS
LIN {X 61.321,Y 94.552,Z 74.500,A 180.000,B 0.000,C 180.000} C_DIS
LIN {X 61.143,Y 94.483,Z 74.500,A 180.000,B 0.000,C 180.000} C_DIS
LIN {X 60.785,Y 94.360,Z 74.500,A 180.000,B 0.000,C 180.000} C_DIS
LIN {X 60.606,Y 94.302,Z 74.500,A 180.000,B 0.000,C 180.000} C_DIS
LIN {X 60.427,Y 94.256,Z 74.500,A 180.000,B 0.000,C 180.000} C_DIS
LIN {X 60.249,Y 94.212,Z 74.500,A 180.000,B 0.000,C 180.000} C_DIS
LIN {X 60.070,Y 94.167,Z 74.500,A 180.000,B 0.000,C 180.000} C_DIS
LIN {X 59.891,Y 94.131,Z 74.500,A 180.000,B 0.000,C 180.000} C_DIS
LIN {X 59.712,Y 94.103,Z 74.500,A 180.000,B 0.000,C 180.000} C_DIS
LIN {X 59.534,Y 94.075,Z 74.500,A 180.000,B 0.000,C 180.000} C_DIS
LIN {X 59.355,Y 94.049,Z 74.500,A 180.000,B 0.000,C 180.000} C_DIS
LIN {X 59.220,Y 94.036,Z 74.500,A 180.000,B 0.000,C 180.000} C_DIS
LIN {X 58.819,Y 94.010,Z 74.500,A 180.000,B 0.000,C 180.000} C_DIS
LIN {X 58.640,Y 94.001,Z 74.500,A 180.000,B 0.000,C 180.000} C_DIS
LIN {X 58.461,Y 94.004,Z 74.500,A 180.000,B 0.000,C 180.000} C_DIS
LIN {X 58.282,Y 94.008,Z 74.500,A 180.000,B 0.000,C 180.000} C_DIS
LIN {X 58.103,Y 94.012,Z 74.500,A 180.000,B 0.000,C 180.000} C_DIS
LIN {X 57.925,Y 94.023,Z 74.500,A 180.000,B 0.000,C 180.000} C_DIS
LIN {X 57.803,Y 94.036,Z 74.500,A 180.000,B 0.000,C 180.000} C_DIS
LIN {X 57.567,Y 94.062,Z 74.500,A 180.000,B 0.000,C 180.000} C_DIS
LIN {X 57.388,Y 94.083,Z 74.500,A 180.000,B 0.000,C 180.000} C_DIS
LIN {X 57.210,Y 94.114,Z 74.500,A 180.000,B 0.000,C 180.000} C_DIS
LIN {X 56.852,Y 94.186,Z 74.500,A 180.000,B 0.000,C 180.000} C_DIS
LIN {X 56.717,Y 94.215,Z 74.500,A 180.000,B 0.000,C 180.000} C_DIS
LIN {X 56.673,Y 94.226,Z 74.500,A 180.000,B 0.000,C 180.000} C_DIS
LIN {X 56.495,Y 94.277,Z 74.500,A 180.000,B 0.000,C 180.000} C_DIS
LIN {X 56.316,Y 94.330,Z 74.500,A 180.000,B 0.000,C 180.000} C_DIS
LIN {X 56.137,Y 94.383,Z 74.500,A 180.000,B 0.000,C 180.000} C_DIS
LIN {X 56.103,Y 94.394,Z 74.500,A 180.000,B 0.000,C 180.000} C_DIS
LIN {X 55.958,Y 94.445,Z 74.500,A 180.000,B 0.000,C 180.000} C_DIS
LIN {X 55.601,Y 94.587,Z 74.500,A 180.000,B 0.000,C 180.000} C_DIS
LIN {X 55.422,Y 94.661,Z 74.500,A 180.000,B 0.000,C 180.000} C_DIS
LIN {X 55.243,Y 94.749,Z 74.500,A 180.000,B 0.000,C 180.000} C_DIS
LIN {X 55.064,Y 94.838,Z 74.500,A 180.000,B 0.000,C 180.000} C_DIS
LIN {X 54.886,Y 94.929,Z 74.500,A 180.000,B 0.000,C 180.000} C_DIS
LIN {X 54.883,Y 94.930,Z 74.500,A 180.000,B 0.000,C 180.000} C_DIS
LIN {X 54.707,Y 95.033,Z 74.500,A 180.000,B 0.000,C 180.000} C_DIS
LIN {X 54.528,Y 95.144,Z 74.500,A 180.000,B 0.000,C 180.000} C_DIS
LIN {X 54.349,Y 95.254,Z 74.500,A 180.000,B 0.000,C 180.000} C_DIS
LIN {X 54.298,Y 95.288,Z 74.500,A 180.000,B 0.000,C 180.000} C_DIS
LIN {X 54.171,Y 95.379,Z 74.500,A 180.000,B 0.000,C 180.000} C_DIS
LIN {X 53.992,Y 95.512,Z 74.500,A 180.000,B 0.000,C 180.000} C_DIS
LIN {X 53.814,Y 95.645,Z 74.500,A 180.000,B 0.000,C 180.000} C_DIS
LIN {X 53.813,Y 95.646,Z 74.500,A 180.000,B 0.000,C 180.000} C_DIS
LIN {X 53.634,Y 95.796,Z 74.500,A 180.000,B 0.000,C 180.000} C_DIS
LIN {X 53.404,Y 96.003,Z 74.500,A 180.000,B 0.000,C 180.000} C_DIS
LIN {X 53.277,Y 96.118,Z 74.500,A 180.000,B 0.000,C 180.000} C_DIS
LIN {X 53.213,Y 96.181,Z 74.500,A 180.000,B 0.000,C 180.000} C_DIS
LIN {X 53.098,Y 96.303,Z 74.500,A 180.000,B 0.000,C 180.000} C_DIS
LIN {X 52.877,Y 96.539,Z 74.500,A 180.000,B 0.000,C 180.000} C_DIS
LIN {X 52.740,Y 96.698,Z 74.500,A 180.000,B 0.000,C 180.000} C_DIS
LIN {X 52.725,Y 96.718,Z 74.500,A 180.000,B 0.000,C 180.000} C_DIS
LIN {X 52.562,Y 96.927,Z 74.500,A 180.000,B 0.000,C 180.000} C_DIS
LIN {X 52.446,Y 97.075,Z 74.500,A 180.000,B 0.000,C 180.000} C_DIS
LIN {X 52.383,Y 97.161,Z 74.500,A 180.000,B 0.000,C 180.000} C_DIS
LIN {X 52.320,Y 97.254,Z 74.500,A 180.000,B 0.000,C 180.000} C_DIS
LIN {X 52.088,Y 97.612,Z 74.500,A 180.000,B 0.000,C 180.000} C_DIS
LIN {X 52.025,Y 97.715,Z 74.500,A 180.000,B 0.000,C 180.000} C_DIS
LIN {X 51.983,Y 97.790,Z 74.500,A 180.000,B 0.000,C 180.000} C_DIS
LIN {X 51.889,Y 97.969,Z 74.500,A 180.000,B 0.000,C 180.000} C_DIS
LIN {X 51.794,Y 98.148,Z 74.500,A 180.000,B 0.000,C 180.000} C_DIS
LIN {X 51.705,Y 98.327,Z 74.500,A 180.000,B 0.000,C 180.000} C_DIS
LIN {X 51.668,Y 98.412,Z 74.500,A 180.000,B 0.000,C 180.000} C_DIS
LIN {X 51.553,Y 98.684,Z 74.500,A 180.000,B 0.000,C 180.000} C_DIS
LIN {X 51.489,Y 98.838,Z 74.500,A 180.000,B 0.000,C 180.000} C_DIS
LIN {X 51.479,Y 98.863,Z 74.500,A 180.000,B 0.000,C 180.000} C_DIS
LIN {X 51.417,Y 99.042,Z 74.500,A 180.000,B 0.000,C 180.000} C_DIS
LIN {X 51.303,Y 99.399,Z 74.500,A 180.000,B 0.000,C 180.000} C_DIS
LIN {X 51.251,Y 99.578,Z 74.500,A 180.000,B 0.000,C 180.000} C_DIS
LIN {X 51.210,Y 99.757,Z 74.500,A 180.000,B 0.000,C 180.000} C_DIS
LIN {X 51.170,Y 99.936,Z 74.500,A 180.000,B 0.000,C 180.000} C_DIS
LIN {X 51.131,Y 100.106,Z 74.500,A 180.000,B 0.000,C 180.000} C_DIS
LIN {X 51.130,Y 100.114,Z 74.500,A 180.000,B 0.000,C 180.000} C_DIS
LIN {X 51.100,Y 100.293,Z 74.500,A 180.000,B 0.000,C 180.000} C_DIS
LIN {X 51.052,Y 100.651,Z 74.500,A 180.000,B 0.000,C 180.000} C_DIS
LIN {X 51.030,Y 100.829,Z 74.500,A 180.000,B 0.000,C 180.000} C_DIS
LIN {X 51.019,Y 101.008,Z 74.500,A 180.000,B 0.000,C 180.000} C_DIS
LIN {X 51.003,Y 101.366,Z 74.500,A 180.000,B 0.000,C 180.000} C_DIS
LIN {X 51.000,Y 101.545,Z 74.500,A 180.000,B 0.000,C 180.000} C_DIS
LIN {X 51.007,Y 101.723,Z 74.500,A 180.000,B 0.000,C 180.000} C_DIS
LIN {X 51.015,Y 101.902,Z 74.500,A 180.000,B 0.000,C 180.000} C_DIS
LIN {X 51.023,Y 102.081,Z 74.500,A 180.000,B 0.000,C 180.000} C_DIS
LIN {X 51.040,Y 102.260,Z 74.500,A 180.000,B 0.000,C 180.000} C_DIS
LIN {X 51.064,Y 102.438,Z 74.500,A 180.000,B 0.000,C 180.000} C_DIS
LIN {X 51.088,Y 102.617,Z 74.500,A 180.000,B 0.000,C 180.000} C_DIS
LIN {X 51.113,Y 102.796,Z 74.500,A 180.000,B 0.000,C 180.000} C_DIS
LIN {X 51.131,Y 102.894,Z 74.500,A 180.000,B 0.000,C 180.000} C_DIS
LIN {X 51.149,Y 102.975,Z 74.500,A 180.000,B 0.000,C 180.000} C_DIS
LIN {X 51.230,Y 103.332,Z 74.500,A 180.000,B 0.000,C 180.000} C_DIS
LIN {X 51.275,Y 103.511,Z 74.500,A 180.000,B 0.000,C 180.000} C_DIS
LIN {X 51.310,Y 103.624,Z 74.500,A 180.000,B 0.000,C 180.000} C_DIS
LIN {X 51.388,Y 103.869,Z 74.500,A 180.000,B 0.000,C 180.000} C_DIS
LIN {X 51.446,Y 104.047,Z 74.500,A 180.000,B 0.000,C 180.000} C_DIS
LIN {X 51.489,Y 104.162,Z 74.500,A 180.000,B 0.000,C 180.000} C_DIS
LIN {X 51.515,Y 104.226,Z 74.500,A 180.000,B 0.000,C 180.000} C_DIS
LIN {X 51.668,Y 104.588,Z 74.500,A 180.000,B 0.000,C 180.000} C_DIS
LIN {X 51.747,Y 104.762,Z 74.500,A 180.000,B 0.000,C 180.000} C_DIS
LIN {X 51.841,Y 104.941,Z 74.500,A 180.000,B 0.000,C 180.000} C_DIS
LIN {X 51.936,Y 105.120,Z 74.500,A 180.000,B 0.000,C 180.000} C_DIS
LIN {X 52.025,Y 105.285,Z 74.500,A 180.000,B 0.000,C 180.000} C_DIS
LIN {X 52.033,Y 105.299,Z 74.500,A 180.000,B 0.000,C 180.000} C_DIS
LIN {X 52.146,Y 105.477,Z 74.500,A 180.000,B 0.000,C 180.000} C_DIS
LIN {X 52.262,Y 105.656,Z 74.500,A 180.000,B 0.000,C 180.000} C_DIS
LIN {X 52.380,Y 105.835,Z 74.500,A 180.000,B 0.000,C 180.000} C_DIS
LIN {X 52.383,Y 105.839,Z 74.500,A 180.000,B 0.000,C 180.000} C_DIS
LIN {X 52.515,Y 106.014,Z 74.500,A 180.000,B 0.000,C 180.000} C_DIS
LIN {X 52.655,Y 106.193,Z 74.500,A 180.000,B 0.000,C 180.000} C_DIS
LIN {X 52.740,Y 106.302,Z 74.500,A 180.000,B 0.000,C 180.000} C_DIS
LIN {X 52.797,Y 106.371,Z 74.500,A 180.000,B 0.000,C 180.000} C_DIS
LIN {X 52.919,Y 106.506,Z 74.500,A 180.000,B 0.000,C 180.000} C_DIS
LIN {X 53.128,Y 106.729,Z 74.500,A 180.000,B 0.000,C 180.000} C_DIS
LIN {X 53.226,Y 106.829,Z 74.500,A 180.000,B 0.000,C 180.000} C_DIS
LIN {X 53.277,Y 106.882,Z 74.500,A 180.000,B 0.000,C 180.000} C_DIS
LIN {X 53.304,Y 106.908,Z 74.500,A 180.000,B 0.000,C 180.000} C_DIS
LIN {X 53.455,Y 107.044,Z 74.500,A 180.000,B 0.000,C 180.000} C_DIS
LIN {X 53.634,Y 107.204,Z 74.500,A 180.000,B 0.000,C 180.000} C_DIS
LIN {X 53.704,Y 107.265,Z 74.500,A 180.000,B 0.000,C 180.000} C_DIS
LIN {X 53.813,Y 107.354,Z 74.500,A 180.000,B 0.000,C 180.000} C_DIS
LIN {X 53.933,Y 107.444,Z 74.500,A 180.000,B 0.000,C 180.000} C_DIS
LIN {X 54.172,Y 107.623,Z 74.500,A 180.000,B 0.000,C 180.000} C_DIS
LIN {X 54.349,Y 107.746,Z 74.500,A 180.000,B 0.000,C 180.000} C_DIS
LIN {X 54.439,Y 107.802,Z 74.500,A 180.000,B 0.000,C 180.000} C_DIS
LIN {X 54.729,Y 107.980,Z 74.500,A 180.000,B 0.000,C 180.000} C_DIS
LIN {X 54.886,Y 108.071,Z 74.500,A 180.000,B 0.000,C 180.000} C_DIS
LIN {X 55.059,Y 108.159,Z 74.500,A 180.000,B 0.000,C 180.000} C_DIS
LIN {X 55.243,Y 108.251,Z 74.500,A 180.000,B 0.000,C 180.000} C_DIS
LIN {X 55.419,Y 108.338,Z 74.500,A 180.000,B 0.000,C 180.000} C_DIS
LIN {X 55.422,Y 108.339,Z 74.500,A 180.000,B 0.000,C 180.000} C_DIS
LIN {X 55.601,Y 108.413,Z 74.500,A 180.000,B 0.000,C 180.000} C_DIS
LIN {X 55.862,Y 108.517,Z 74.500,A 180.000,B 0.000,C 180.000} C_DIS
LIN {X 55.958,Y 108.555,Z 74.500,A 180.000,B 0.000,C 180.000} C_DIS
LIN {X 56.137,Y 108.617,Z 74.500,A 180.000,B 0.000,C 180.000} C_DIS
LIN {X 56.316,Y 108.670,Z 74.500,A 180.000,B 0.000,C 180.000} C_DIS
LIN {X 56.495,Y 108.723,Z 74.500,A 180.000,B 0.000,C 180.000} C_DIS
LIN {X 56.673,Y 108.774,Z 74.500,A 180.000,B 0.000,C 180.000} C_DIS
LIN {X 56.852,Y 108.814,Z 74.500,A 180.000,B 0.000,C 180.000} C_DIS
LIN {X 57.210,Y 108.886,Z 74.500,A 180.000,B 0.000,C 180.000} C_DIS
LIN {X 57.388,Y 108.917,Z 74.500,A 180.000,B 0.000,C 180.000} C_DIS
LIN {X 57.567,Y 108.938,Z 74.500,A 180.000,B 0.000,C 180.000} C_DIS
LIN {X 57.746,Y 108.957,Z 74.500,A 180.000,B 0.000,C 180.000} C_DIS
LIN {X 57.925,Y 108.977,Z 74.500,A 180.000,B 0.000,C 180.000} C_DIS
LIN {X 58.103,Y 108.988,Z 74.500,A 180.000,B 0.000,C 180.000} C_DIS
LIN {X 58.282,Y 108.992,Z 74.500,A 180.000,B 0.000,C 180.000} C_DIS
LIN {X 58.461,Y 108.996,Z 74.500,A 180.000,B 0.000,C 180.000} C_DIS
LIN {X 58.640,Y 108.999,Z 74.500,A 180.000,B 0.000,C 180.000} C_DIS
LIN {X 58.819,Y 108.990,Z 74.500,A 180.000,B 0.000,C 180.000} C_DIS
LIN {X 59.176,Y 108.967,Z 74.500,A 180.000,B 0.000,C 180.000} C_DIS
LIN {X 59.355,Y 108.951,Z 74.500,A 180.000,B 0.000,C 180.000} C_DIS
LIN {X 59.534,Y 108.925,Z 74.500,A 180.000,B 0.000,C 180.000} C_DIS
LIN {X 59.856,Y 108.874,Z 74.500,A 180.000,B 0.000,C 180.000} C_DIS
LIN {X 59.891,Y 108.869,Z 74.500,A 180.000,B 0.000,C 180.000} C_DIS
LIN {X 60.070,Y 108.833,Z 74.500,A 180.000,B 0.000,C 180.000} C_DIS
LIN {X 60.249,Y 108.788,Z 74.500,A 180.000,B 0.000,C 180.000} C_DIS
LIN {X 60.427,Y 108.744,Z 74.500,A 180.000,B 0.000,C 180.000} C_DIS
LIN {X 60.606,Y 108.698,Z 74.500,A 180.000,B 0.000,C 180.000} C_DIS
LIN {X 60.616,Y 108.695,Z 74.500,A 180.000,B 0.000,C 180.000} C_DIS
LIN {X 60.785,Y 108.640,Z 74.500,A 180.000,B 0.000,C 180.000} C_DIS
LIN {X 61.144,Y 108.517,Z 74.500,A 180.000,B 0.000,C 180.000} C_DIS
LIN {X 61.321,Y 108.448,Z 74.500,A 180.000,B 0.000,C 180.000} C_DIS
LIN {X 61.500,Y 108.369,Z 74.500,A 180.000,B 0.000,C 180.000} C_DIS
LIN {X 61.679,Y 108.289,Z 74.500,A 180.000,B 0.000,C 180.000} C_DIS
LIN {X 61.858,Y 108.206,Z 74.500,A 180.000,B 0.000,C 180.000} C_DIS
LIN {X 61.948,Y 108.159,Z 74.500,A 180.000,B 0.000,C 180.000} C_DIS
LIN {X 62.036,Y 108.110,Z 74.500,A 180.000,B 0.000,C 180.000} C_DIS
LIN {X 62.268,Y 107.980,Z 74.500,A 180.000,B 0.000,C 180.000} C_DIS
LIN {X 62.394,Y 107.909,Z 74.500,A 180.000,B 0.000,C 180.000} C_DIS
LIN {X 62.562,Y 107.802,Z 74.500,A 180.000,B 0.000,C 180.000} C_DIS
LIN {X 62.825,Y 107.623,Z 74.500,A 180.000,B 0.000,C 180.000} C_DIS
LIN {X 62.930,Y 107.551,Z 74.500,A 180.000,B 0.000,C 180.000} C_DIS
LIN {X 63.071,Y 107.444,Z 74.500,A 180.000,B 0.000,C 180.000} C_DIS
LIN {X 63.109,Y 107.413,Z 74.500,A 180.000,B 0.000,C 180.000} C_DIS
LIN {X 63.290,Y 107.265,Z 74.500,A 180.000,B 0.000,C 180.000} C_DIS
LIN {X 63.467,Y 107.120,Z 74.500,A 180.000,B 0.000,C 180.000} C_DIS
LIN {X 63.504,Y 107.086,Z 74.500,A 180.000,B 0.000,C 180.000} C_DIS
LIN {X 63.645,Y 106.952,Z 74.500,A 180.000,B 0.000,C 180.000} C_DIS
LIN {X 63.873,Y 106.729,Z 74.500,A 180.000,B 0.000,C 180.000} C_DIS
LIN {X 64.003,Y 106.596,Z 74.500,A 180.000,B 0.000,C 180.000} C_DIS
LIN {X 64.043,Y 106.550,Z 74.500,A 180.000,B 0.000,C 180.000} C_DIS
LIN {X 64.196,Y 106.371,Z 74.500,A 180.000,B 0.000,C 180.000} C_DIS
LIN {X 64.349,Y 106.193,Z 74.500,A 180.000,B 0.000,C 180.000} C_DIS
LIN {X 64.360,Y 106.179,Z 74.500,A 180.000,B 0.000,C 180.000} C_DIS
LIN {X 64.487,Y 106.014,Z 74.500,A 180.000,B 0.000,C 180.000} C_DIS
LIN {X 64.718,Y 105.690,Z 74.500,A 180.000,B 0.000,C 180.000} C_DIS
LIN {X 64.742,Y 105.656,Z 74.500,A 180.000,B 0.000,C 180.000} C_DIS
LIN {X 64.856,Y 105.477,Z 74.500,A 180.000,B 0.000,C 180.000} C_DIS
LIN {X 65.075,Y 105.104,Z 74.500,A 180.000,B 0.000,C 180.000} C_DIS
LIN {X 65.163,Y 104.941,Z 74.500,A 180.000,B 0.000,C 180.000} C_DIS
LIN {X 65.248,Y 104.762,Z 74.500,A 180.000,B 0.000,C 180.000} C_DIS
LIN {X 65.333,Y 104.584,Z 74.500,A 180.000,B 0.000,C 180.000} C_DIS
LIN {X 65.415,Y 104.405,Z 74.500,A 180.000,B 0.000,C 180.000} C_DIS
LIN {X 65.433,Y 104.360,Z 74.500,A 180.000,B 0.000,C 180.000} C_DIS
LIN {X 65.483,Y 104.226,Z 74.500,A 180.000,B 0.000,C 180.000} C_DIS
LIN {X 65.549,Y 104.047,Z 74.500,A 180.000,B 0.000,C 180.000} C_DIS
LIN {X 65.612,Y 103.878,Z 74.500,A 180.000,B 0.000,C 180.000} C_DIS
LIN {X 65.615,Y 103.869,Z 74.500,A 180.000,B 0.000,C 180.000} C_DIS
LIN {X 65.672,Y 103.690,Z 74.500,A 180.000,B 0.000,C 180.000} C_DIS
LIN {X 65.720,Y 103.511,Z 74.500,A 180.000,B 0.000,C 180.000} C_DIS
LIN {X 65.791,Y 103.253,Z 74.500,A 180.000,B 0.000,C 180.000} C_DIS
LIN {X 65.815,Y 103.153,Z 74.500,A 180.000,B 0.000,C 180.000} C_DIS
LIN {X 65.850,Y 102.975,Z 74.500,A 180.000,B 0.000,C 180.000} C_DIS
LIN {X 65.914,Y 102.617,Z 74.500,A 180.000,B 0.000,C 180.000} C_DIS
LIN {X 65.941,Y 102.438,Z 74.500,A 180.000,B 0.000,C 180.000} C_DIS
LIN {X 65.957,Y 102.260,Z 74.500,A 180.000,B 0.000,C 180.000} C_DIS
LIN {X 65.973,Y 102.081,Z 74.500,A 180.000,B 0.000,C 180.000} C_DIS
LIN {X 65.989,Y 101.902,Z 74.500,A 180.000,B 0.000,C 180.000} C_DIS
LIN {X 65.995,Y 101.723,Z 74.500,A 180.000,B 0.000,C 180.000} C_DIS
LIN {X 65.995,Y 101.366,Z 74.500,A 180.000,B 0.000,C 180.000} C_DIS
LIN {X 65.993,Y 101.187,Z 74.500,A 180.000,B 0.000,C 180.000} C_DIS
LIN {X 65.981,Y 101.008,Z 74.500,A 180.000,B 0.000,C 180.000} C_DIS
LIN {X 65.949,Y 100.651,Z 74.500,A 180.000,B 0.000,C 180.000} C_DIS
LIN {X 65.942,Y 100.588,Z 74.500,A 180.000,B 0.000,C 180.000} C_DIS
; Link Move Starts
LIN {X 65.973,Y 100.430,Z 74.500,A 180.000,B 0.000,C 180.000} C_DIS
LIN {X 65.945,Y 100.271,Z 74.500,A 180.000,B 0.000,C 180.000} C_DIS
LIN {X 65.890,Y 99.961,Z 74.499,A 180.000,B 0.000,C 180.000} C_DIS
LIN {X 65.858,Y 99.807,Z 74.498,A 180.000,B 0.000,C 180.000} C_DIS
LIN {X 65.817,Y 99.655,Z 74.498,A 180.000,B 0.000,C 180.000} C_DIS
LIN {X 65.735,Y 99.351,Z 74.496,A 180.000,B 0.000,C 180.000} C_DIS
LIN {X 65.691,Y 99.200,Z 74.495,A 180.000,B 0.000,C 180.000} C_DIS
LIN {X 65.639,Y 99.051,Z 74.494,A 180.000,B 0.000,C 180.000} C_DIS
LIN {X 65.530,Y 98.756,Z 74.492,A 180.000,B 0.000,C 180.000} C_DIS
LIN {X 65.474,Y 98.608,Z 74.490,A 180.000,B 0.000,C 180.000} C_DIS
LIN {X 65.411,Y 98.464,Z 74.489,A 180.000,B 0.000,C 180.000} C_DIS
LIN {X 65.276,Y 98.179,Z 74.485,A 180.000,B 0.000,C 180.000} C_DIS
LIN {X 65.134,Y 97.898,Z 74.481,A 180.000,B 0.000,C 180.000} C_DIS
LIN {X 64.975,Y 97.626,Z 74.477,A 180.000,B 0.000,C 180.000} C_DIS
LIN {X 64.811,Y 97.357,Z 74.472,A 180.000,B 0.000,C 180.000} C_DIS
LIN {X 64.721,Y 97.228,Z 74.470,A 180.000,B 0.000,C 180.000} C_DIS
LIN {X 64.629,Y 97.100,Z 74.467,A 180.000,B 0.000,C 180.000} C_DIS
LIN {X 64.538,Y 96.972,Z 74.465,A 180.000,B 0.000,C 180.000} C_DIS
LIN {X 64.444,Y 96.845,Z 74.462,A 180.000,B 0.000,C 180.000} C_DIS
LIN {X 64.344,Y 96.724,Z 74.459,A 180.000,B 0.000,C 180.000} C_DIS
LIN {X 64.241,Y 96.604,Z 74.456,A 180.000,B 0.000,C 180.000} C_DIS
LIN {X 64.139,Y 96.485,Z 74.453,A 180.000,B 0.000,C 180.000} C_DIS
LIN {X 64.035,Y 96.366,Z 74.450,A 180.000,B 0.000,C 180.000} C_DIS
LIN {X 63.926,Y 96.253,Z 74.447,A 180.000,B 0.000,C 180.000} C_DIS
LIN {X 63.813,Y 96.143,Z 74.443,A 180.000,B 0.000,C 180.000} C_DIS
LIN {X 63.700,Y 96.032,Z 74.440,A 180.000,B 0.000,C 180.000} C_DIS
LIN {X 63.588,Y 95.923,Z 74.436,A 180.000,B 0.000,C 180.000} C_DIS
LIN {X 63.470,Y 95.818,Z 74.433,A 180.000,B 0.000,C 180.000} C_DIS
LIN {X 63.348,Y 95.718,Z 74.429,A 180.000,B 0.000,C 180.000} C_DIS
LIN {X 63.226,Y 95.618,Z 74.426,A 180.000,B 0.000,C 180.000} C_DIS
LIN {X 63.104,Y 95.519,Z 74.422,A 180.000,B 0.000,C 180.000} C_DIS
LIN {X 62.979,Y 95.423,Z 74.418,A 180.000,B 0.000,C 180.000} C_DIS
LIN {X 62.850,Y 95.334,Z 74.414,A 180.000,B 0.000,C 180.000} C_DIS
LIN {X 62.719,Y 95.245,Z 74.410,A 180.000,B 0.000,C 180.000} C_DIS
LIN {X 62.589,Y 95.156,Z 74.406,A 180.000,B 0.000,C 180.000} C_DIS
LIN {X 62.457,Y 95.070,Z 74.401,A 180.000,B 0.000,C 180.000} C_DIS
LIN {X 62.321,Y 94.992,Z 74.397,A 180.000,B 0.000,C 180.000} C_DIS
LIN {X 62.183,Y 94.915,Z 74.393,A 180.000,B 0.000,C 180.000} C_DIS
LIN {X 62.046,Y 94.838,Z 74.388,A 180.000,B 0.000,C 180.000} C_DIS
LIN {X 61.907,Y 94.763,Z 74.384,A 180.000,B 0.000,C 180.000} C_DIS
LIN {X 61.765,Y 94.695,Z 74.379,A 180.000,B 0.000,C 180.000} C_DIS
LIN {X 61.621,Y 94.631,Z 74.375,A 180.000,B 0.000,C 180.000} C_DIS
LIN {X 61.478,Y 94.566,Z 74.370,A 180.000,B 0.000,C 180.000} C_DIS
LIN {X 61.334,Y 94.503,Z 74.365,A 180.000,B 0.000,C 180.000} C_DIS
LIN {X 61.187,Y 94.446,Z 74.360,A 180.000,B 0.000,C 180.000} C_DIS
LIN {X 61.038,Y 94.394,Z 74.355,A 180.000,B 0.000,C 180.000} C_DIS
LIN {X 60.815,Y 94.317,Z 74.348,A 180.000,B 0.000,C 180.000} C_DIS
LIN {X 60.740,Y 94.292,Z 74.345,A 180.000,B 0.000,C 180.000} C_DIS
LIN {X 60.665,Y 94.267,Z 74.343,A 180.000,B 0.000,C 180.000} C_DIS
LIN {X 60.590,Y 94.245,Z 74.340,A 180.000,B 0.000,C 180.000} C_DIS
LIN {X 60.513,Y 94.226,Z 74.338,A 180.000,B 0.000,C 180.000} C_DIS
LIN {X 60.437,Y 94.207,Z 74.335,A 180.000,B 0.000,C 180.000} C_DIS
LIN {X 60.284,Y 94.169,Z 74.330,A 180.000,B 0.000,C 180.000} C_DIS
LIN {X 60.131,Y 94.131,Z 74.325,A 180.000,B 0.000,C 180.000} C_DIS
LIN {X 60.055,Y 94.112,Z 74.322,A 180.000,B 0.000,C 180.000} C_DIS
LIN {X 59.978,Y 94.096,Z 74.319,A 180.000,B 0.000,C 180.000} C_DIS
LIN {X 59.900,Y 94.082,Z 74.317,A 180.000,B 0.000,C 180.000} C_DIS
LIN {X 59.822,Y 94.070,Z 74.314,A 180.000,B 0.000,C 180.000} C_DIS
LIN {X 59.667,Y 94.046,Z 74.308,A 180.000,B 0.000,C 180.000} C_DIS
LIN {X 59.511,Y 94.021,Z 74.303,A 180.000,B 0.000,C 180.000} C_DIS
LIN {X 59.433,Y 94.009,Z 74.300,A 180.000,B 0.000,C 180.000} C_DIS
LIN {X 59.355,Y 93.999,Z 74.297,A 180.000,B 0.000,C 180.000} C_DIS
LIN {X 59.277,Y 93.991,Z 74.295,A 180.000,B 0.000,C 180.000} C_DIS
LIN {X 59.198,Y 93.985,Z 74.292,A 180.000,B 0.000,C 180.000} C_DIS
LIN {X 58.963,Y 93.969,Z 74.284,A 180.000,B 0.000,C 180.000} C_DIS
LIN {X 58.805,Y 93.959,Z 74.278,A 180.000,B 0.000,C 180.000} C_DIS
LIN {X 58.727,Y 93.954,Z 74.275,A 180.000,B 0.000,C 180.000} C_DIS
LIN {X 58.648,Y 93.951,Z 74.273,A 180.000,B 0.000,C 180.000} C_DIS
LIN {X 58.569,Y 93.952,Z 74.270,A 180.000,B 0.000,C 180.000} C_DIS
LIN {X 58.491,Y 93.953,Z 74.267,A 180.000,B 0.000,C 180.000} C_DIS
LIN {X 58.412,Y 93.955,Z 74.264,A 180.000,B 0.000,C 180.000} C_DIS
LIN {X 58.254,Y 93.959,Z 74.259,A 180.000,B 0.000,C 180.000} C_DIS
LIN {X 58.176,Y 93.960,Z 74.256,A 180.000,B 0.000,C 180.000} C_DIS
LIN {X 58.097,Y 93.962,Z 74.253,A 180.000,B 0.000,C 180.000} C_DIS
LIN {X 58.018,Y 93.965,Z 74.251,A 180.000,B 0.000,C 180.000} C_DIS
LIN {X 57.940,Y 93.971,Z 74.248,A 180.000,B 0.000,C 180.000} C_DIS
LIN {X 57.861,Y 93.979,Z 74.245,A 180.000,B 0.000,C 180.000} C_DIS
LIN {X 57.783,Y 93.988,Z 74.242,A 180.000,B 0.000,C 180.000} C_DIS
LIN {X 57.627,Y 94.006,Z 74.237,A 180.000,B 0.000,C 180.000} C_DIS
LIN {X 57.470,Y 94.023,Z 74.231,A 180.000,B 0.000,C 180.000} C_DIS
LIN {X 57.392,Y 94.032,Z 74.229,A 180.000,B 0.000,C 180.000} C_DIS
LIN {X 57.314,Y 94.044,Z 74.226,A 180.000,B 0.000,C 180.000} C_DIS
LIN {X 57.236,Y 94.058,Z 74.223,A 180.000,B 0.000,C 180.000} C_DIS
LIN {X 57.159,Y 94.073,Z 74.220,A 180.000,B 0.000,C 180.000} C_DIS
LIN {X 57.005,Y 94.105,Z 74.215,A 180.000,B 0.000,C 180.000} C_DIS
LIN {X 56.850,Y 94.136,Z 74.209,A 180.000,B 0.000,C 180.000} C_DIS
LIN {X 56.773,Y 94.151,Z 74.207,A 180.000,B 0.000,C 180.000} C_DIS
LIN {X 56.696,Y 94.169,Z 74.204,A 180.000,B 0.000,C 180.000} C_DIS
LIN {X 56.620,Y 94.188,Z 74.201,A 180.000,B 0.000,C 180.000} C_DIS
LIN {X 56.545,Y 94.210,Z 74.198,A 180.000,B 0.000,C 180.000} C_DIS
LIN {X 56.393,Y 94.255,Z 74.193,A 180.000,B 0.000,C 180.000} C_DIS
LIN {X 56.167,Y 94.322,Z 74.185,A 180.000,B 0.000,C 180.000} C_DIS
LIN {X 56.092,Y 94.345,Z 74.182,A 180.000,B 0.000,C 180.000} C_DIS
LIN {X 56.017,Y 94.370,Z 74.179,A 180.000,B 0.000,C 180.000} C_DIS
LIN {X 55.943,Y 94.398,Z 74.176,A 180.000,B 0.000,C 180.000} C_DIS
LIN {X 55.797,Y 94.455,Z 74.171,A 180.000,B 0.000,C 180.000} C_DIS
LIN {X 55.577,Y 94.542,Z 74.163,A 180.000,B 0.000,C 180.000} C_DIS
LIN {X 55.504,Y 94.571,Z 74.160,A 180.000,B 0.000,C 180.000} C_DIS
LIN {X 55.431,Y 94.602,Z 74.157,A 180.000,B 0.000,C 180.000} C_DIS
LIN {X 55.360,Y 94.635,Z 74.154,A 180.000,B 0.000,C 180.000} C_DIS
LIN {X 55.289,Y 94.670,Z 74.152,A 180.000,B 0.000,C 180.000} C_DIS
LIN {X 54.937,Y 94.846,Z 74.138,A 180.000,B 0.000,C 180.000} C_DIS
LIN {X 54.867,Y 94.882,Z 74.135,A 180.000,B 0.000,C 180.000} C_DIS
LIN {X 54.798,Y 94.920,Z 74.132,A 180.000,B 0.000,C 180.000} C_DIS
LIN {X 54.730,Y 94.960,Z 74.130,A 180.000,B 0.000,C 180.000} C_DIS
LIN {X 54.462,Y 95.126,Z 74.119,A 180.000,B 0.000,C 180.000} C_DIS
LIN {X 54.395,Y 95.167,Z 74.116,A 180.000,B 0.000,C 180.000} C_DIS
LIN {X 54.328,Y 95.209,Z 74.113,A 180.000,B 0.000,C 180.000} C_DIS
LIN {X 54.262,Y 95.251,Z 74.110,A 180.000,B 0.000,C 180.000} C_DIS
LIN {X 54.198,Y 95.297,Z 74.108,A 180.000,B 0.000,C 180.000} C_DIS
LIN {X 54.134,Y 95.343,Z 74.105,A 180.000,B 0.000,C 180.000} C_DIS
LIN {X 53.819,Y 95.579,Z 74.091,A 180.000,B 0.000,C 180.000} C_DIS
LIN {X 53.756,Y 95.627,Z 74.089,A 180.000,B 0.000,C 180.000} C_DIS
LIN {X 53.695,Y 95.676,Z 74.086,A 180.000,B 0.000,C 180.000} C_DIS
LIN {X 53.636,Y 95.728,Z 74.083,A 180.000,B 0.000,C 180.000} C_DIS
LIN {X 53.342,Y 95.991,Z 74.069,A 180.000,B 0.000,C 180.000} C_DIS
LIN {X 53.284,Y 96.043,Z 74.067,A 180.000,B 0.000,C 180.000} C_DIS
LIN {X 53.226,Y 96.097,Z 74.064,A 180.000,B 0.000,C 180.000} C_DIS
LIN {X 53.171,Y 96.153,Z 74.061,A 180.000,B 0.000,C 180.000} C_DIS
LIN {X 53.117,Y 96.210,Z 74.058,A 180.000,B 0.000,C 180.000} C_DIS
LIN {X 52.848,Y 96.498,Z 74.045,A 180.000,B 0.000,C 180.000} C_DIS
LIN {X 52.794,Y 96.556,Z 74.042,A 180.000,B 0.000,C 180.000} C_DIS
LIN {X 52.743,Y 96.616,Z 74.039,A 180.000,B 0.000,C 180.000} C_DIS
LIN {X 52.694,Y 96.677,Z 74.036,A 180.000,B 0.000,C 180.000} C_DIS
LIN {X 52.451,Y 96.987,Z 74.023,A 180.000,B 0.000,C 180.000} C_DIS
LIN {X 52.403,Y 97.049,Z 74.020,A 180.000,B 0.000,C 180.000} C_DIS
LIN {X 52.356,Y 97.112,Z 74.017,A 180.000,B 0.000,C 180.000} C_DIS
LIN {X 52.311,Y 97.177,Z 74.014,A 180.000,B 0.000,C 180.000} C_DIS
LIN {X 52.268,Y 97.243,Z 74.012,A 180.000,B 0.000,C 180.000} C_DIS
LIN {X 52.054,Y 97.574,Z 73.998,A 180.000,B 0.000,C 180.000} C_DIS
LIN {X 52.012,Y 97.640,Z 73.995,A 180.000,B 0.000,C 180.000} C_DIS
LIN {X 51.972,Y 97.708,Z 73.992,A 180.000,B 0.000,C 180.000} C_DIS
LIN {X 51.934,Y 97.777,Z 73.990,A 180.000,B 0.000,C 180.000} C_DIS
LIN {X 51.750,Y 98.125,Z 73.976,A 180.000,B 0.000,C 180.000} C_DIS
LIN {X 51.713,Y 98.195,Z 73.973,A 180.000,B 0.000,C 180.000} C_DIS
LIN {X 51.678,Y 98.265,Z 73.970,A 180.000,B 0.000,C 180.000} C_DIS
LIN {X 51.645,Y 98.337,Z 73.968,A 180.000,B 0.000,C 180.000} C_DIS
LIN {X 51.615,Y 98.410,Z 73.965,A 180.000,B 0.000,C 180.000} C_DIS
LIN {X 51.462,Y 98.772,Z 73.951,A 180.000,B 0.000,C 180.000} C_DIS
LIN {X 51.432,Y 98.845,Z 73.948,A 180.000,B 0.000,C 180.000} C_DIS
LIN {X 51.405,Y 98.919,Z 73.946,A 180.000,B 0.000,C 180.000} C_DIS
LIN {X 51.380,Y 98.994,Z 73.943,A 180.000,B 0.000,C 180.000} C_DIS
LIN {X 51.260,Y 99.369,Z 73.929,A 180.000,B 0.000,C 180.000} C_DIS
LIN {X 51.236,Y 99.444,Z 73.926,A 180.000,B 0.000,C 180.000} C_DIS
LIN {X 51.214,Y 99.520,Z 73.924,A 180.000,B 0.000,C 180.000} C_DIS
LIN {X 51.195,Y 99.596,Z 73.921,A 180.000,B 0.000,C 180.000} C_DIS
LIN {X 51.177,Y 99.673,Z 73.918,A 180.000,B 0.000,C 180.000} C_DIS
LIN {X 51.091,Y 100.057,Z 73.904,A 180.000,B 0.000,C 180.000} C_DIS
LIN {X 51.075,Y 100.134,Z 73.902,A 180.000,B 0.000,C 180.000} C_DIS
LIN {X 51.061,Y 100.212,Z 73.899,A 180.000,B 0.000,C 180.000} C_DIS
LIN {X 51.050,Y 100.290,Z 73.896,A 180.000,B 0.000,C 180.000} C_DIS
LIN {X 50.997,Y 100.680,Z 73.882,A 180.000,B 0.000,C 180.000} C_DIS
LIN {X 50.987,Y 100.758,Z 73.880,A 180.000,B 0.000,C 180.000} C_DIS
LIN {X 50.979,Y 100.836,Z 73.877,A 180.000,B 0.000,C 180.000} C_DIS
LIN {X 50.974,Y 100.915,Z 73.874,A 180.000,B 0.000,C 180.000} C_DIS
LIN {X 50.970,Y 100.994,Z 73.871,A 180.000,B 0.000,C 180.000} C_DIS
LIN {X 50.963,Y 101.151,Z 73.866,A 180.000,B 0.000,C 180.000} C_DIS
LIN {X 50.953,Y 101.387,Z 73.858,A 180.000,B 0.000,C 180.000} C_DIS
LIN {X 50.950,Y 101.466,Z 73.855,A 180.000,B 0.000,C 180.000} C_DIS
LIN {X 50.950,Y 101.544,Z 73.852,A 180.000,B 0.000,C 180.000} C_DIS
LIN {X 50.953,Y 101.623,Z 73.849,A 180.000,B 0.000,C 180.000} C_DIS
LIN {X 50.960,Y 101.780,Z 73.844,A 180.000,B 0.000,C 180.000} C_DIS
LIN {X 50.970,Y 102.016,Z 73.836,A 180.000,B 0.000,C 180.000} C_DIS
LIN {X 50.974,Y 102.095,Z 73.833,A 180.000,B 0.000,C 180.000} C_DIS
LIN {X 50.980,Y 102.174,Z 73.830,A 180.000,B 0.000,C 180.000} C_DIS
LIN {X 50.989,Y 102.252,Z 73.827,A 180.000,B 0.000,C 180.000} C_DIS
LIN {X 50.999,Y 102.330,Z 73.825,A 180.000,B 0.000,C 180.000} C_DIS
LIN {X 51.020,Y 102.486,Z 73.819,A 180.000,B 0.000,C 180.000} C_DIS
LIN {X 51.051,Y 102.720,Z 73.811,A 180.000,B 0.000,C 180.000} C_DIS
LIN {X 51.063,Y 102.798,Z 73.808,A 180.000,B 0.000,C 180.000} C_DIS
LIN {X 51.077,Y 102.876,Z 73.805,A 180.000,B 0.000,C 180.000} C_DIS
LIN {X 51.093,Y 102.953,Z 73.803,A 180.000,B 0.000,C 180.000} C_DIS
LIN {X 51.128,Y 103.106,Z 73.797,A 180.000,B 0.000,C 180.000} C_DIS
LIN {X 51.180,Y 103.337,Z 73.789,A 180.000,B 0.000,C 180.000} C_DIS
LIN {X 51.197,Y 103.414,Z 73.786,A 180.000,B 0.000,C 180.000} C_DIS
LIN {X 51.217,Y 103.490,Z 73.783,A 180.000,B 0.000,C 180.000} C_DIS
LIN {X 51.239,Y 103.565,Z 73.781,A 180.000,B 0.000,C 180.000} C_DIS
LIN {X 51.263,Y 103.640,Z 73.778,A 180.000,B 0.000,C 180.000} C_DIS
LIN {X 51.311,Y 103.790,Z 73.772,A 180.000,B 0.000,C 180.000} C_DIS
LIN {X 51.335,Y 103.865,Z 73.770,A 180.000,B 0.000,C 180.000} C_DIS
LIN {X 51.383,Y 104.015,Z 73.764,A 180.000,B 0.000,C 180.000} C_DIS
LIN {X 51.408,Y 104.090,Z 73.761,A 180.000,B 0.000,C 180.000} C_DIS
LIN {X 51.436,Y 104.164,Z 73.759,A 180.000,B 0.000,C 180.000} C_DIS
LIN {X 51.466,Y 104.237,Z 73.756,A 180.000,B 0.000,C 180.000} C_DIS
LIN {X 51.527,Y 104.382,Z 73.750,A 180.000,B 0.000,C 180.000} C_DIS
LIN {X 51.557,Y 104.454,Z 73.748,A 180.000,B 0.000,C 180.000} C_DIS
LIN {X 51.618,Y 104.600,Z 73.742,A 180.000,B 0.000,C 180.000} C_DIS
LIN {X 51.649,Y 104.672,Z 73.739,A 180.000,B 0.000,C 180.000} C_DIS
LIN {X 51.682,Y 104.744,Z 73.737,A 180.000,B 0.000,C 180.000} C_DIS
LIN {X 51.717,Y 104.814,Z 73.734,A 180.000,B 0.000,C 180.000} C_DIS
LIN {X 51.754,Y 104.884,Z 73.731,A 180.000,B 0.000,C 180.000} C_DIS
LIN {X 51.865,Y 105.093,Z 73.723,A 180.000,B 0.000,C 180.000} C_DIS
LIN {X 51.938,Y 105.232,Z 73.717,A 180.000,B 0.000,C 180.000} C_DIS
LIN {X 51.977,Y 105.301,Z 73.715,A 180.000,B 0.000,C 180.000} C_DIS
LIN {X 52.017,Y 105.368,Z 73.712,A 180.000,B 0.000,C 180.000} C_DIS
LIN {X 52.059,Y 105.435,Z 73.709,A 180.000,B 0.000,C 180.000} C_DIS
LIN {X 52.188,Y 105.633,Z 73.701,A 180.000,B 0.000,C 180.000} C_DIS
LIN {X 52.273,Y 105.765,Z 73.695,A 180.000,B 0.000,C 180.000} C_DIS
LIN {X 52.316,Y 105.831,Z 73.693,A 180.000,B 0.000,C 180.000} C_DIS
LIN {X 52.362,Y 105.896,Z 73.690,A 180.000,B 0.000,C 180.000} C_DIS
LIN {X 52.409,Y 105.959,Z 73.687,A 180.000,B 0.000,C 180.000} C_DIS
LIN {X 52.457,Y 106.021,Z 73.684,A 180.000,B 0.000,C 180.000} C_DIS
LIN {X 52.554,Y 106.145,Z 73.679,A 180.000,B 0.000,C 180.000} C_DIS
LIN {X 52.651,Y 106.269,Z 73.674,A 180.000,B 0.000,C 180.000} C_DIS
LIN {X 52.700,Y 106.331,Z 73.671,A 180.000,B 0.000,C 180.000} C_DIS
LIN {X 52.749,Y 106.392,Z 73.668,A 180.000,B 0.000,C 180.000} C_DIS
LIN {X 52.801,Y 106.452,Z 73.666,A 180.000,B 0.000,C 180.000} C_DIS
LIN {X 52.854,Y 106.509,Z 73.663,A 180.000,B 0.000,C 180.000} C_DIS
LIN {X 52.962,Y 106.624,Z 73.658,A 180.000,B 0.000,C 180.000} C_DIS
LIN {X 53.016,Y 106.682,Z 73.655,A 180.000,B 0.000,C 180.000} C_DIS
LIN {X 53.070,Y 106.739,Z 73.653,A 180.000,B 0.000,C 180.000} C_DIS
LIN {X 53.123,Y 106.797,Z 73.650,A 180.000,B 0.000,C 180.000} C_DIS
LIN {X 53.233,Y 106.910,Z 73.645,A 180.000,B 0.000,C 180.000} C_DIS
LIN {X 53.350,Y 107.016,Z 73.640,A 180.000,B 0.000,C 180.000} C_DIS
LIN {X 53.467,Y 107.121,Z 73.636,A 180.000,B 0.000,C 180.000} C_DIS
LIN {X 53.584,Y 107.226,Z 73.631,A 180.000,B 0.000,C 180.000} C_DIS
LIN {X 53.703,Y 107.330,Z 73.626,A 180.000,B 0.000,C 180.000} C_DIS
LIN {X 53.827,Y 107.427,Z 73.621,A 180.000,B 0.000,C 180.000} C_DIS
LIN {X 53.953,Y 107.521,Z 73.617,A 180.000,B 0.000,C 180.000} C_DIS
LIN {X 54.079,Y 107.615,Z 73.612,A 180.000,B 0.000,C 180.000} C_DIS
LIN {X 54.206,Y 107.709,Z 73.608,A 180.000,B 0.000,C 180.000} C_DIS
LIN {X 54.337,Y 107.797,Z 73.603,A 180.000,B 0.000,C 180.000} C_DIS
LIN {X 54.471,Y 107.880,Z 73.599,A 180.000,B 0.000,C 180.000} C_DIS
LIN {X 54.605,Y 107.962,Z 73.595,A 180.000,B 0.000,C 180.000} C_DIS
LIN {X 54.739,Y 108.045,Z 73.591,A 180.000,B 0.000,C 180.000} C_DIS
LIN {X 54.876,Y 108.123,Z 73.587,A 180.000,B 0.000,C 180.000} C_DIS
LIN {X 55.016,Y 108.194,Z 73.583,A 180.000,B 0.000,C 180.000} C_DIS
LIN {X 55.157,Y 108.264,Z 73.579,A 180.000,B 0.000,C 180.000} C_DIS
LIN {X 55.298,Y 108.335,Z 73.575,A 180.000,B 0.000,C 180.000} C_DIS
LIN {X 55.440,Y 108.402,Z 73.571,A 180.000,B 0.000,C 180.000} C_DIS
LIN {X 55.586,Y 108.461,Z 73.567,A 180.000,B 0.000,C 180.000} C_DIS
LIN {X 55.733,Y 108.519,Z 73.564,A 180.000,B 0.000,C 180.000} C_DIS
LIN {X 55.879,Y 108.577,Z 73.560,A 180.000,B 0.000,C 180.000} C_DIS
LIN {X 56.026,Y 108.633,Z 73.557,A 180.000,B 0.000,C 180.000} C_DIS
LIN {X 56.177,Y 108.681,Z 73.554,A 180.000,B 0.000,C 180.000} C_DIS
LIN {X 56.328,Y 108.726,Z 73.550,A 180.000,B 0.000,C 180.000} C_DIS
LIN {X 56.479,Y 108.770,Z 73.547,A 180.000,B 0.000,C 180.000} C_DIS
LIN {X 56.630,Y 108.814,Z 73.544,A 180.000,B 0.000,C 180.000} C_DIS
LIN {X 56.783,Y 108.851,Z 73.541,A 180.000,B 0.000,C 180.000} C_DIS
LIN {X 56.937,Y 108.882,Z 73.538,A 180.000,B 0.000,C 180.000} C_DIS
LIN {X 57.092,Y 108.913,Z 73.535,A 180.000,B 0.000,C 180.000} C_DIS
LIN {X 57.246,Y 108.944,Z 73.533,A 180.000,B 0.000,C 180.000} C_DIS
LIN {X 57.402,Y 108.969,Z 73.530,A 180.000,B 0.000,C 180.000} C_DIS
LIN {X 57.558,Y 108.987,Z 73.528,A 180.000,B 0.000,C 180.000} C_DIS
LIN {X 57.871,Y 109.022,Z 73.523,A 180.000,B 0.000,C 180.000} C_DIS
LIN {X 58.028,Y 109.035,Z 73.521,A 180.000,B 0.000,C 180.000} C_DIS
LIN {X 58.186,Y 109.040,Z 73.519,A 180.000,B 0.000,C 180.000} C_DIS
LIN {X 58.501,Y 109.047,Z 73.515,A 180.000,B 0.000,C 180.000} C_DIS
LIN {X 58.658,Y 109.048,Z 73.513,A 180.000,B 0.000,C 180.000} C_DIS
LIN {X 58.815,Y 109.041,Z 73.511,A 180.000,B 0.000,C 180.000} C_DIS
LIN {X 59.130,Y 109.020,Z 73.508,A 180.000,B 0.000,C 180.000} C_DIS
LIN {X 59.287,Y 109.009,Z 73.507,A 180.000,B 0.000,C 180.000} C_DIS
LIN {X 59.443,Y 108.989,Z 73.506,A 180.000,B 0.000,C 180.000} C_DIS
LIN {X 59.754,Y 108.941,Z 73.504,A 180.000,B 0.000,C 180.000} C_DIS
LIN {X 60.064,Y 108.885,Z 73.502,A 180.000,B 0.000,C 180.000} C_DIS
LIN {X 60.370,Y 108.810,Z 73.501,A 180.000,B 0.000,C 180.000} C_DIS
LIN {X 60.675,Y 108.730,Z 73.500,A 180.000,B 0.000,C 180.000} C_DIS
LIN {X 60.958,Y 108.633,Z 73.500,A 180.000,B 0.000,C 180.000} C_DIS
; Cutting Move Starts
LIN {X 61.143,Y 108.570,Z 73.500,A 180.000,B 0.000,C 180.000} C_DIS
LIN {X 61.287,Y 108.517,Z 73.500,A 180.000,B 0.000,C 180.000} C_DIS
